CASE fb_state_entry.i16_step OF
(*=======================================================*)
	0:	(* *)
		st_ecd_cmd.enu_cmd := NO_COMMAND;
		st_ecd_cmd.b_job_fehler := FALSE;
		mc_gearindyn_axis.Enable := FALSE;
		mc_gearout_axis.Execute := FALSE;
		mc_camin_axis.Execute := FALSE;
		mc_camout_axis.Execute := FALSE;
		mc_cam_scaleing.Execute := FALSE;
		mc_read_motion_function_point.Execute := FALSE;
		mc_write_motion_function_point.Execute := FALSE;
		mc_read_camtable_slave_dynamics.Execute := FALSE;
		mc_read_camtable_characteristics.Execute := FALSE;
		st_ecd_cmd.meldungen.sm_gear_in_slave := FALSE;
		st_ecd_cmd.meldungen.sm_gear_out_slave := FALSE;
		st_ecd_cmd.meldungen.sm_cam_in_slave := FALSE;
		st_ecd_cmd.meldungen.sm_cam_out_slave := FALSE;
		st_ecd_cmd.meldungen.sm_cam_scaleing_slave := FALSE;
		st_ecd_cmd.meldungen.sm_write_motion_funktion_point := FALSE;
		st_ecd_cmd.meldungen.sm_read_motion_funktion_point := FALSE;
		st_ecd_cmd.meldungen.sm_read_camtable_slave_dynamics := FALSE;
		st_ecd_cmd.meldungen.sm_read_camtable_charakteristik := FALSE;
		st_ecd_cmd.meldungen.sm_camgear_command_timeout := FALSE;

		fb_ton_cmd_timeout.IN := FALSE;
		fb_state_entry.i16_next_step := 10;

(*=======================================================*)
	10:	(* Warte auf Kommando *)
		IF fb_state_entry.E THEN
			st_ecd_cmd.b_job_fehler := FALSE;
			st_ecd_cmd.enu_cmd := NO_COMMAND;
		END_IF

		IF st_ecd_cmd.enu_cmd > NO_COMMAND THEN
			(* Diese Kommandos werden mit Direktsprung ausgeführt, um Zykluszeit zu sparen *)
			IF st_ecd_cmd.enu_cmd = GEAR_IN_SLAVE THEN
				fb_state_entry.i16_next_step := 20;
			ELSIF st_ecd_cmd.enu_cmd = GEAR_OUT_SLAVE THEN
				fb_state_entry.i16_next_step := 30;
			ELSIF st_ecd_cmd.enu_cmd = CAM_IN_SLAVE THEN
				fb_state_entry.i16_next_step := 40;
			ELSIF st_ecd_cmd.enu_cmd = CAM_OUT_SLAVE THEN
				fb_state_entry.i16_next_step := 50;
			ELSIF st_ecd_cmd.enu_cmd = CAM_SCALEING_SLAVE THEN
				fb_state_entry.i16_next_step := 60;
			ELSIF st_ecd_cmd.enu_cmd = READ_MOTION_POINT THEN
				fb_state_entry.i16_next_step := 70;
			ELSIF st_ecd_cmd.enu_cmd = WRITE_MOTION_POINT THEN
				fb_state_entry.i16_next_step := 80;
			ELSIF st_ecd_cmd.enu_cmd = READ_SLAVE_DYNAMICS THEN
				fb_state_entry.i16_next_step := 90;
			ELSIF st_ecd_cmd.enu_cmd = READ_CAMTABLE_CHAR THEN
				fb_state_entry.i16_next_step := 100;
			ELSIF st_ecd_cmd.enu_cmd = RESET THEN
				fb_state_entry.i16_next_step := 999;
			ELSE
				fb_state_entry.i16_next_step := 1000;
			END_IF
		END_IF

(*=======================================================*)
	20:	(* Gear in *)
		fb_ton_cmd_timeout.IN := TRUE;
		mc_gearindyn_axis.Enable := TRUE;
		IF mc_gearindyn_axis.Busy THEN
			fb_state_entry.i16_next_step := 22;
		END_IF

	22:
		IF mc_gearindyn_axis.InGear THEN
			mc_gearindyn_axis.Enable := FALSE;
			fb_state_entry.i16_next_step := 999;
		ELSIF mc_gearindyn_axis.Error THEN
			st_ecd_cmd.meldungen.sm_gear_in_slave := TRUE;
			err_id := mc_gearindyn_axis.ErrorID;
			fb_state_entry.i16_next_step := 1000;
		END_IF

		IF st_ecd_cmd.enu_cmd = GEAR_OUT_SLAVE THEN
			mc_gearindyn_axis.Enable := FALSE;
			fb_ton_cmd_timeout.IN := FALSE;
			fb_ton_vz.IN := FALSE;
			fb_state_entry.i16_next_step := 50;
		END_IF

(*=======================================================*)
	30:	(* Gear out *)
		fb_ton_cmd_timeout.IN := TRUE;
		mc_gearout_axis.Execute := TRUE;
		IF mc_gearout_axis.Busy THEN
			fb_state_entry.i16_next_step := 32;
		END_IF
	32:
		IF NOT mc_gearout_axis.Busy THEN
			mc_gearout_axis.Execute := FALSE;
			IF mc_gearout_axis.Done THEN
				fb_state_entry.i16_next_step := 999;
			ELSIF mc_gearout_axis.Error THEN
				st_ecd_cmd.meldungen.sm_gear_out_slave := TRUE;
				err_id := mc_gearout_axis.ErrorID;
				fb_state_entry.i16_next_step := 1000;
			END_IF
		END_IF

(*=======================================================*)
	40:	(* Cam in *)
		fb_ton_cmd_timeout.IN := NOT st_slaveachse.Status.CamTableQueued;
		mc_camin_axis.Execute := TRUE;
		IF mc_camin_axis.Busy THEN
			fb_state_entry.i16_next_step := 42;
		END_IF
		IF st_ecd_cmd.enu_cmd = CAM_OUT_SLAVE THEN
			mc_camin_axis.Execute := FALSE;
			fb_state_entry.i16_next_step := 50;
		END_IF
	42:
		fb_ton_cmd_timeout.IN := NOT st_slaveachse.Status.CamTableQueued;
		IF NOT mc_camin_axis.Busy THEN
			mc_camin_axis.Execute := FALSE;
			IF mc_camin_axis.InSync THEN
				fb_state_entry.i16_next_step := 999;
			ELSIF mc_camin_axis.Error THEN
				err_id := mc_camin_axis.ErrorID;
				mc_camin_axis.Execute := FALSE;
				st_ecd_cmd.meldungen.sm_cam_in_slave := TRUE;
				fb_state_entry.i16_next_step := 1000;
			END_IF
		END_IF

		IF st_ecd_cmd.enu_cmd = CAM_OUT_SLAVE THEN
			mc_camin_axis.Execute := FALSE;
			fb_ton_cmd_timeout.IN := FALSE;
			fb_ton_vz.IN := FALSE;
			fb_state_entry.i16_next_step := 50;
		END_IF

(*=======================================================*)
	50:	(* Cam out *)
		fb_ton_cmd_timeout.IN := TRUE;
		mc_camout_axis.Execute := TRUE;
		IF mc_camout_axis.Busy THEN
			fb_state_entry.i16_next_step := 52;
		END_IF
	52:
		IF NOT mc_camout_axis.Busy THEN
			mc_camout_axis.Execute := FALSE;
			IF mc_camout_axis.Done THEN
				fb_state_entry.i16_next_step := 999;
			ELSIF mc_camout_axis.Error THEN
				st_ecd_cmd.meldungen.sm_cam_out_slave := TRUE;
				err_id := mc_camout_axis.ErrorID;
				fb_state_entry.i16_next_step := 1000;
			END_IF
		END_IF

(*=======================================================*)
	60:	(* Cam scaleing *)
		fb_ton_cmd_timeout.IN := NOT st_slaveachse.Status.CamScalingPending;
		mc_cam_scaleing.Execute := TRUE;
		IF mc_cam_scaleing.Busy THEN
			fb_state_entry.i16_next_step := 62;
		END_IF
	62:
		fb_ton_cmd_timeout.IN := NOT st_slaveachse.Status.CamScalingPending;
		IF NOT mc_cam_scaleing.Busy THEN
			mc_cam_scaleing.Execute := FALSE;
			IF mc_cam_scaleing.Done THEN
				fb_state_entry.i16_next_step := 999;
			ELSIF mc_cam_scaleing.Error THEN
				st_ecd_cmd.meldungen.sm_cam_scaleing_slave := TRUE;
				err_id := mc_cam_scaleing.ErrorID;
				fb_state_entry.i16_next_step := 1000;
			END_IF
		END_IF

		IF st_ecd_cmd.enu_cmd = CAM_OUT_SLAVE THEN
			mc_cam_scaleing.Execute := FALSE;
			fb_ton_cmd_timeout.IN := FALSE;
			fb_ton_vz.IN := FALSE;
			fb_state_entry.i16_next_step := 50;
		END_IF

(*=======================================================*)
	70:	(* Lesen Motion Funktion Point *)
		fb_ton_cmd_timeout.IN := TRUE;
		mc_read_motion_function_point.Execute := TRUE;
		IF mc_read_motion_function_point.Busy THEN
			fb_state_entry.i16_next_step := 72;
		END_IF
	72:
		IF NOT mc_read_motion_function_point.Busy THEN
			mc_read_motion_function_point.Execute := FALSE;
			IF mc_read_motion_function_point.Done THEN
				fb_state_entry.i16_next_step := 999;
			ELSIF mc_read_motion_function_point.Error THEN
				st_ecd_cmd.meldungen.sm_read_motion_funktion_point := TRUE;
				err_id := mc_read_motion_function_point.ErrorID;
				fb_state_entry.i16_next_step := 1000;
			END_IF
		END_IF

(*=======================================================*)
	80:	(* Schreiben Motion Funktion Point *)
		fb_ton_cmd_timeout.IN := TRUE;
		mc_write_motion_function_point.Execute := TRUE;
		IF mc_write_motion_function_point.Busy THEN
			fb_state_entry.i16_next_step := 82;
		END_IF
	82:
		IF NOT mc_write_motion_function_point.Busy THEN
			mc_write_motion_function_point.Execute := FALSE;
			IF mc_write_motion_function_point.Done THEN
				fb_state_entry.i16_next_step := 999;
			ELSIF mc_write_motion_function_point.Error THEN
				st_ecd_cmd.meldungen.sm_write_motion_funktion_point := TRUE;
				err_id := mc_write_motion_function_point.ErrorID;
				fb_state_entry.i16_next_step := 1000;
			END_IF
		END_IF

(*=======================================================*)
	90:	(* Lesen der Slaveposition in einer Kurvenscheibe *)
		fb_ton_cmd_timeout.IN := TRUE;
		mc_read_camtable_slave_dynamics.Execute := TRUE;
		IF mc_read_camtable_slave_dynamics.Busy THEN
			fb_state_entry.i16_next_step := 92;
		END_IF
	92:
		IF NOT mc_read_camtable_slave_dynamics.Busy THEN
			mc_read_camtable_slave_dynamics.Execute := FALSE;
			IF mc_read_camtable_slave_dynamics.Done THEN
				fb_state_entry.i16_next_step := 999;
			ELSIF mc_read_camtable_slave_dynamics.Error THEN
				st_ecd_cmd.meldungen.sm_write_motion_funktion_point := TRUE;
				err_id := mc_read_camtable_slave_dynamics.ErrorID;
				fb_state_entry.i16_next_step := 1000;
			END_IF
		END_IF

(*=======================================================*)
	100:	(* Lesen der charakteristischen Werte einer Kurvenscheibe *)
		fb_ton_cmd_timeout.IN := TRUE;
		mc_read_camtable_characteristics.Execute := TRUE;
		IF mc_read_camtable_characteristics.Busy THEN
			fb_state_entry.i16_next_step := 102;
		END_IF
	102:
		IF NOT mc_read_camtable_characteristics.Busy THEN
			mc_read_camtable_characteristics.Execute := FALSE;
			IF mc_read_camtable_characteristics.Done THEN
				fb_state_entry.i16_next_step := 999;
			ELSIF mc_read_camtable_characteristics.Error THEN
				st_ecd_cmd.meldungen.sm_read_camtable_charakteristik := TRUE;
				err_id := mc_read_camtable_slave_dynamics.ErrorID;
				fb_state_entry.i16_next_step := 1000;
			END_IF
		END_IF

(*=======================================================*)
	999:	(* Ende - Befehl wurde korrekt abgearbeitet *)
		fb_ton_cmd_timeout.IN := FALSE;
		fb_ton_vz.IN := FALSE;

		mc_gearindyn_axis.Enable := FALSE;
		mc_gearout_axis.Execute := FALSE;
		mc_camin_axis.Execute := FALSE;
		mc_camout_axis.Execute := FALSE;
		mc_cam_scaleing.Execute := FALSE;
		mc_read_motion_function_point.Execute := FALSE;
		mc_write_motion_function_point.Execute := FALSE;
		mc_read_camtable_slave_dynamics.Execute := FALSE;
		mc_read_camtable_characteristics.Execute := FALSE;

		st_ecd_cmd.meldungen.sm_gear_in_slave := FALSE;
		st_ecd_cmd.meldungen.sm_gear_out_slave := FALSE;
		st_ecd_cmd.meldungen.sm_cam_in_slave := FALSE;
		st_ecd_cmd.meldungen.sm_cam_out_slave := FALSE;
		st_ecd_cmd.meldungen.sm_cam_scaleing_slave := FALSE;
		st_ecd_cmd.meldungen.sm_write_motion_funktion_point := FALSE;
		st_ecd_cmd.meldungen.sm_read_motion_funktion_point := FALSE;
		st_ecd_cmd.meldungen.sm_read_camtable_slave_dynamics := FALSE;
		st_ecd_cmd.meldungen.sm_read_camtable_charakteristik := FALSE;
		st_ecd_cmd.meldungen.sm_camgear_command_timeout := FALSE;

		fb_state_entry.i16_next_step := 10;

(*=======================================================*)
	1000: (* Fehler *)
		IF fb_state_entry.E THEN
			st_ecd_cmd.enu_cmd := NO_COMMAND;
			st_ecd_cmd.b_job_fehler := TRUE;
			fb_ton_cmd_timeout.IN := FALSE;
			fb_ton_vz.IN := FALSE;

			mc_gearindyn_axis.Enable := FALSE;
			mc_gearout_axis.Execute := FALSE;
			mc_camin_axis.Execute := FALSE;
			mc_camout_axis.Execute := FALSE;
			mc_cam_scaleing.Execute := FALSE;
			mc_read_motion_function_point.Execute := FALSE;
			mc_write_motion_function_point.Execute := FALSE;
			mc_read_camtable_slave_dynamics.Execute := FALSE;
			mc_read_camtable_characteristics.Execute := FALSE;
		END_IF

		(* Fehler reseten *)
		IF st_ecd_cmd.enu_cmd > ABORT THEN
			st_ecd_cmd.b_job_fehler := FALSE;

			st_ecd_cmd.meldungen.sm_gear_in_slave := FALSE;
			st_ecd_cmd.meldungen.sm_gear_out_slave := FALSE;
			st_ecd_cmd.meldungen.sm_cam_in_slave := FALSE;
			st_ecd_cmd.meldungen.sm_cam_out_slave := FALSE;
			st_ecd_cmd.meldungen.sm_cam_scaleing_slave := FALSE;
			st_ecd_cmd.meldungen.sm_write_motion_funktion_point := FALSE;
			st_ecd_cmd.meldungen.sm_read_motion_funktion_point := FALSE;
			st_ecd_cmd.meldungen.sm_read_camtable_slave_dynamics := FALSE;
			st_ecd_cmd.meldungen.sm_read_camtable_charakteristik := FALSE;
			st_ecd_cmd.meldungen.sm_camgear_command_timeout := FALSE;

			fb_state_entry.i16_next_step := 10;
			err_id :=0;
		END_IF
END_CASE

(* Timeout-Fehler aller Drivekommandos *)
IF fb_ton_cmd_timeout.Q THEN
	fb_ton_cmd_timeout.IN := FALSE;
	st_ecd_cmd.meldungen.sm_camgear_command_timeout := TRUE;
	fb_state_entry.i16_next_step := 1000;
END_IF

(* Statehistory *)
fb_state_entry(
	i16_next_step:= , 
	i16_pos:= 2,
	s_debugtext:= ,
	E=> ,
	X=> , 
	i16_step=> ,
	i16_last_step=> );

fb_cmd_history(i16_current_cmd:= st_ecd_cmd.enu_cmd, last_cmd=> );

(*=============================================================================================*)
(* Ab hier werden alle Cam und Gear Aufträge für eine Achse abgewickelt *)

(* Getriebegleichlauf an der Slaveachse einschalten *)
(* Alternativ kann der Getriebefaktor im Zähler als Fließkommawert angegeben werden, wenn der Nenner 1 ist. *)
mc_gearindyn_axis(
	Enable:= , 
	GearRatio:= r_getriebefaktor,
	Acceleration:= , 
	Deceleration:= , 
	Jerk:= , 
	BufferMode:= mc_buffermode_axis,
	Options:= , 
	Master:= st_masterachse,
	Slave:= st_slaveachse,
	InGear=> , 
	Busy=> , 
	Active=> , 
	CommandAborted=> , 
	Error=> , 
	ErrorID=> );

(*=============================================================================================*)
(* Getriebegleichlauf ausschalten *)
mc_gearout_axis(
	Execute:= ,
	Options:= ,
	Slave:= st_slaveachse,
	Done=> ,
	Busy=> ,
	Error=> ,
	ErrorID=> );

(*=============================================================================================*)
(* Kurvenscheibe am Slave aktivieren *)
mc_camin_axis(
	Execute:= , 
	ActivationMode:= mc_activation_mode_camin,
	ActivationPosition:= lr_activation_position_camin,
	CamTableID:= mc_cam_table_id,
	Scaling:= st_camscaling_data,
	Options:= st_camin_options,
	Master:= st_masterachse,
	Slave:= st_slaveachse,
	InSync=> , 
	Busy=> , 
	Active=> , 
	CommandAborted=> , 
	Error=> ,
	ErrorID=> );

(*=============================================================================================*)
(* Kurvenscheibe ausschalten *)
mc_camout_axis(
	Execute:= ,
	Slave:= st_slaveachse,
	Options:= ,
	Done=> ,
	Busy=> ,
	Error=> ,
	ErrorID=> );

(*=============================================================================================*)
(* Scalierung einer Kurvenscheibe *)
mc_cam_scaleing(
	Execute:= , 
	ActivationMode:= mc_activation_mode_scaleing,
	ActivationPosition:= lr_activation_position_scaleing,
	CamTableID:= mc_cam_table_id,
	Scaling:= st_camscaling_data,
	Options:= ,
	Slave:= st_slaveachse,
	Done=> , 
	Busy=> ,
	Active=> , 
	CommandAborted=> ,
	Error=> , 
	ErrorID=> );

(*=============================================================================================*)
(* Lesen eines Punktes in der Kurvenscheibe *)
mc_read_motion_function_point(
	Execute:= ,
	CamTableID:= mc_cam_table_id,
	PointID:= mc_cam_point_id,
	Point:= mc_motion_function_point,
	Done=> , 
	Busy=> , 
	Error=> , 
	ErrorID=> );

(*=============================================================================================*)
(* Verändern von einem Punkt in der Kurvenscheibe *)
mc_write_motion_function_point(
	Execute:= , 
	CamTableID:= mc_cam_table_id,
	PointID:= mc_cam_point_id,
	Point:= mc_motion_function_point,
	Done=> , 
	Busy=> , 
	Error=> ,
	ErrorID=> );

(*=============================================================================================*)
(* Lesen einer Slaveposition in der Kurvenscheibe *)
mc_read_camtable_slave_dynamics(
	Execute:= ,
	CamTableID:= mc_cam_table_id,
	MasterPosition:= r_master_position,
	Done=> , 
	Busy=> ,
	Error=> , 
	ErrorID=> ,
	SlavePosition=> , 
	SlaveVelocity=> , 
	SlaveAcceleration=> );

(*=============================================================================================*)
(* Lesen der charakteristischen Werte einer Kurvenscheibe *)
mc_read_camtable_characteristics(
	Execute:= , 
	CamTableID:= mc_cam_table_id,
	CamTableCharac:= st_cam_table_characteristics,
	Done=> , 
	Busy=> , 
	Error=> , 
	ErrorID=> );
END_FUNCTION_BLOCK

(* POU EPT Lib/Funktionsbausteine/ST_BerechnungOverride, ST *)
FUNCTION_BLOCK ST_BerechnungOverride
VAR_INPUT
	i16_betriebsart				: enum_betriebsarten;
	lr_skalierung_slave_achse1		: LREAL;
	lr_skalierung_slave_achse2		: LREAL;
	lr_override_vorgabe			: LREAL;
	lr_faktor						: LREAL;

	lr_FaktorHub				: LREAL;
	lr_HubAuto					: LREAL;
END_VAR
VAR_OUTPUT
	lr_override					: LREAL := 0.0;
END_VAR
VAR
	lr_offset						: LREAL := 100.0;
	tmp_lr_override_slave1		: LREAL := 0.0;
	tmp_lr_override_slave2		: LREAL := 0.0;

	lr_ProzentDerRichtdrehzahl	: LREAL;
	lr_Reduzierung				: LREAL;
END_VAR
(* Funktion zur Berechnung des Override der  Masterachse: y = - faktor * x^2 + offset *)
(* Die Funktion besteht aus einer auf dem Kopf stehenden Parabel, welche um den faktor nach oben verschoben ist *)
(* Aufpassen bei den Nullstellen der Funktion, wenn faktor und offset verändert werden *)

(* Die Anpassung der maximalen Mastergeschwindigkeit an die Verfahrlänge des Slaves wird hier einfach über eine empirisch ermittelte Funktion realisiert *)
(* Eine verbesserte Anpassung stellt die Berechnung der maximalen Mastergeschwindigkeit (ST_MFMaxMasterVelo) im CamEditor dar. *)

tmp_lr_override_slave1 := - lr_faktor * (lr_skalierung_slave_achse1 * lr_skalierung_slave_achse1)  + lr_offset;
tmp_lr_override_slave2 := - lr_faktor * (lr_skalierung_slave_achse2 * lr_skalierung_slave_achse2)  + lr_offset;

IF tmp_lr_override_slave1 < 0.0 THEN
	 tmp_lr_override_slave1 := 0.0;
ELSIF tmp_lr_override_slave1 >= 100.0 THEN
	 tmp_lr_override_slave1 := 100.0;
END_IF
IF tmp_lr_override_slave2 < 0.0 THEN
	 tmp_lr_override_slave2 := 0.0;
ELSIF tmp_lr_override_slave2 >= 100.0 THEN
	 tmp_lr_override_slave2 := 100.0;
END_IF

IF i16_betriebsart = AUTO THEN
	(* Nur wenn der mit der Funktion berechnete Override kleiner ist, als die Vorgabe, dann wird der Funktionswert übernommen *)
	IF 	tmp_lr_override_slave1 < lr_override_vorgabe OR
		tmp_lr_override_slave2 < lr_override_vorgabe THEN

		IF tmp_lr_override_slave1 <= tmp_lr_override_slave2 THEN
			lr_override := tmp_lr_override_slave1;
		ELSIF tmp_lr_override_slave2 < tmp_lr_override_slave1 THEN
			lr_override := tmp_lr_override_slave2;
		ELSE
			lr_override := lr_override_vorgabe;
		END_IF

	ELSE
		lr_override := lr_override_vorgabe;
	END_IF
ELSE
	lr_override := lr_override_vorgabe;
END_IF


(*neue Berechnung==========================================================================*)
(*Reduzierung abhängig von der Nenndrehzahl*)
lr_ProzentDerRichtdrehzahl:=(lr_HubAuto *100)/250;
IF	lr_HubAuto >250 AND
	lr_override_vorgabe > lr_override THEN
	lr_override := 100-((lr_override_vorgabe - lr_override) * (lr_ProzentDerRichtdrehzahl /100)) ;
END_IF

(*nur Reduzieren wenn das Ergebniss kleiner ist als bei der Reduzierung durch die Pin Anzahl*)
lr_Reduzierung:= (lr_override_vorgabe - lr_override)/100;
IF	(1 - lr_Reduzierung) < lr_FaktorHub THEN
	lr_override := lr_override;
ELSE
	lr_override:= 100 * lr_FaktorHub;
END_IF

IF	lr_override > lr_override_vorgabe OR
	lr_override < 0 THEN
	lr_override:= lr_override_vorgabe;
END_IF

(*Beim Einfädeln wird der Override vom Bausstein ST_TippTasten einfach durchgeschleust*)
IF	ST_TippTasten.b_einfaedeln_aktiv OR
	ST_TippTasten.b_initialisierungsphase THEN
	lr_override := lr_override_vorgabe;
END_IF

(*bei Prüfteilen Override fest auf 30% *)
IF	lr_override_vorgabe > 30 AND
	(FIND( gst_datensatz.st_md.s_aktuelle_artikelnummer,'ruef') <> 0 OR FIND( gst_datensatz.st_md.s_aktuelle_artikelnummer,'erth') <> 0)THEN
	lr_override := 30;
END_IF
END_FUNCTION_BLOCK

(* POU Gemeinsamkeiten17xx/Bedienen/ST_TippTasten, ST *)
PROGRAM ST_TippTasten
VAR_INPUT
	(* Geschwindigkeit / Stufe *)
	i16_akt_stufe						: INT := 0;	(* 0-9 *)
	b_initialisierungsphase				: BOOL := FALSE;
	b_einfaedeln_aktiv				: BOOL := FALSE;
END_VAR
VAR_IN_OUT
	st_visu							: struct_visu;
	st_visu_hinten						: struct_visu_hinten;
END_VAR
VAR
	lr_override						: LREAL := 25;
	lr_override_gestuft					: LREAL := 10;
	r_trig_tippen						: R_TRIG;
	r_trig_tippen_einfaedeln			: R_TRIG;
	r_trig_vorgabe					: R_TRIG;
	b_freigabe_override_auto			: BOOL := FALSE;
	fb_r_trig_quittieren					: R_TRIG;
END_VAR

VAR CONSTANT
	lr_override_init_einfaedel			: LREAL := 25;
END_VAR
(* Mit den zeitlichen Impulsen vom Handrad lässt sich der Override aller Achsen verändern. Die Geschwindigkeit wird im "ST_AxisJobCtrl_Motion" limitiert. *)
(* Tipp-Taste *)

r_trig_tippen(
		CLK:=NOT b_einfaedeln_aktiv AND (st_visu.b_tippen_start OR visu_hinten.out.b_start OR ST_Euchner_Handbedienpult.b_Taste_Power),
		Q=> );
r_trig_tippen_einfaedeln(
		CLK:= b_einfaedeln_aktiv AND (st_visu_hinten.out.b_tippen OR ST_Euchner_Handbedienpult.b_Taste_Power),
		Q=> );
r_trig_vorgabe(
		CLK:= st_visu.b_geschwindigkeit_vorgabe, Q=> );

(* Flanken *)
fb_r_trig_quittieren(CLK:= st_visu.b_quittieren OR st_visu_hinten.out.b_quittieren, Q=> );

CASE gi16_betriebsart OF
	AUTO:
		gb_ba_auto_kontroller := TRUE;

		IF r_trig_tippen.Q OR fb_r_trig_quittieren.Q THEN
			b_freigabe_override_auto := TRUE;
		END_IF

		IF b_einfaedeln_aktiv OR b_initialisierungsphase THEN
			lr_override := lr_override_gestuft := lr_override_init_einfaedel;
		ELSE

			IF r_trig_vorgabe.Q THEN
				i16_akt_stufe := 9;
			END_IF
			IF b_freigabe_override_auto THEN
				(* Override für Achsen mit "Vollgas" im Automatikbetrieb *)
				lr_override := 100;
				(* Override für Achsen, welche in Abstufung gefahren werden *)
				IF  i16_akt_stufe>= 0 AND i16_akt_stufe<= 9 THEN
					(* Overridevorgabe im Automatikbetrieb *)
					lr_override_gestuft := (i16_akt_stufe +1) * 10;
				ELSE
					(* Falls Geschwindigkeitsstufe was anderes als 0-9 enthält: Override auf 0: Keine Achse fährt *)
					lr_override_gestuft := 0;
				END_IF
			ELSE
				lr_override := lr_override_gestuft := 0;
			END_IF
		END_IF

	TIPPEN:
		b_freigabe_override_auto := FALSE;

		IF r_trig_tippen.Q OR lr_override > 0 OR  lr_override_gestuft > 0 THEN
			gb_ba_auto_kontroller := TRUE;
		ELSE
			gb_ba_auto_kontroller := FALSE;
		END_IF

		IF ST_Euchner_Handbedienpult.i16_Handrad_delta > 0 THEN
			lr_override := lr_override_gestuft := ABS(ST_Euchner_Handbedienpult.i16_Handrad_delta) * 0.1;
		ELSE
			lr_override := lr_override_gestuft := 0;
		END_IF

	HAND:
		gb_ba_auto_kontroller := FALSE;
		b_freigabe_override_auto := FALSE;
		lr_override := lr_override_gestuft := ABS(ST_Euchner_Handbedienpult.i16_Handrad_delta)* 0.1;
END_CASE

(* Abfrage maximaler Override grösser 100% *)
IF lr_override > 100 THEN
	lr_override := 100;
END_IF
IF lr_override_gestuft > 100 THEN
	lr_override_gestuft := 100;
END_IF
END_PROGRAM

(* POU Gemeinsamkeiten17xx/Bedienen/ST_Euchner_Handbedienpult, ST *)
PROGRAM ST_Euchner_Handbedienpult
VAR
	(* Eingänge von der Hardware *)
	e_Taste_Zustimm			AT %I* : BOOL;
	e_Taste_Plus				AT %I* : BOOL;
	e_Taste_Power			AT %I* : BOOL;
	e_Taste_Minus			AT %I* : BOOL;

	e_i16_Zaehler			AT %I* : INT;

	(* Instanzen *)
	fb_ton					: TON;

	(* Merker *)
	i16_merkpos				: INT := 0;
END_VAR
VAR_OUTPUT
	b_Taste_Zustimm			: BOOL := FALSE;
	b_Taste_Plus				: BOOL := FALSE;
	b_Taste_Power			: BOOL := FALSE;
	b_Taste_Minus			: BOOL := FALSE;

	i16_Handrad_delta		: INT := 0;
END_VAR
(* Tasten *)
b_Taste_Zustimm	:= e_Taste_Zustimm;
b_Taste_Plus	:= e_Taste_Plus;
b_Taste_Power := e_Taste_Power;
b_Taste_Minus := e_Taste_Minus;

(* Generiere Impuls für Delta Zähler *)
fb_ton(IN:= NOT fb_ton.Q , PT:= t#100ms, Q=> , ET=> );

IF fb_ton.Q THEN
	i16_Handrad_delta := e_i16_Zaehler - i16_merkpos;
	i16_merkpos := e_i16_Zaehler;
END_IF
END_PROGRAM

(* POU Rasterfolie/ST_Rasterfolieneinzug, ST *)
PROGRAM ST_Rasterfolieneinzug
VAR_INPUT
	st_config							: struct_config;
	st_ctrl_in							: struct_ctrl_in;
END_VAR
VAR_IN_OUT
	st_visu							: struct_visu;
END_VAR
VAR_OUTPUT
	st_ctrl_out						: struct_ctrl_out;
END_VAR
VAR
	fb_ton_wz						: TON;
	fb_ton_uez						: TON;
	fb_ton_quitt						: TON;
	fb_ton_gls_rafo_vorhanden		: TON;
	fb_tof_gls_rafo_ende			: TOF;
	fb_tof_AbschaltungIonisierung		: TOF;
	fb_r_trig_start						: R_TRIG;
	fb_r_trig_vorschubkontrolle			: R_TRIG;
	fb_f_trig_vorschubkontrolle			: F_TRIG;
	fb_state_entry						: ST_StateEntry;
	i								: INT := 0;
	sm_fehler_rafo_vorschub			: BOOL := FALSE;
	sm_keine_rafo_im_einzug		: BOOL := FALSE;

	e_rasfo_ende						AT %I* : BOOL;
	e_rasfo_vorschubkontrolle			AT %I* : BOOL;
	e_rasfo_rueckzugueberwachung		AT %I* : BOOL;

	(* Ausgang Ionisierung Rasterfolie einschalten *)
	aIonisierungEin				AT %Q* : BOOL;

END_VAR
(* Zeiten *)
fb_ton_wz(IN:= , PT:= , Q=>  , ET=> );
fb_ton_uez(IN:= , PT:= t#1000ms, Q=>  , ET=> );
fb_ton_quitt(IN:= , PT:= t#100ms, Q=> , ET=> );
fb_ton_gls_rafo_vorhanden(IN:= e_rasfo_ende, PT:= T#300ms, Q=> , ET=> );
fb_tof_gls_rafo_ende(IN:= fb_ton_gls_rafo_vorhanden.Q, PT:= T#300ms, Q=> , ET=> );
fb_tof_AbschaltungIonisierung(IN:= fb_state_entry.i16_step = 200, PT:= T#2m, Q=> , ET=> );

(* Flanken *)
fb_r_trig_start(CLK:= st_ctrl_in.b_start, Q=> );
fb_r_trig_vorschubkontrolle(CLK:= e_rasfo_vorschubkontrolle, Q=> );
fb_f_trig_vorschubkontrolle(CLK:= e_rasfo_vorschubkontrolle, Q=> );


(* Steuerung Ionisierung *)
IF gi16_maschinenstatusinfo = STATUS_MASCHINE_ARBEITET THEN
	aIonisierungEin := fb_tof_AbschaltungIonisierung.Q;
ELSE
	aIonisierungEin := FALSE;
END_IF


(* Toplevel *)
IF fb_state_entry.i16_next_step > INIT AND fb_state_entry.i16_next_step < FEHLER THEN
	IF fb_state_entry.i16_next_step < STOP THEN
		IF st_ctrl_in.b_stop THEN
			fb_state_entry.i16_next_step := STOP;
		END_IF
	END_IF
	(* Allgemeine Fehler *)
	IF	zyl_rafo_faenger.st_ctrl.out.b_fehler OR
		zyl_rafo_klemmen.st_ctrl.out.b_fehler OR
		zyl_rafo_vorschub.st_ctrl.out.b_fehler
		THEN
			fb_state_entry.i16_next_step := FEHLER;

	(* Zylinder im Handbetrieb *)
	ELSIF	gi16_betriebsart = HAND AND (
			(st_visu.st_zyl.i16_nr_zyl_im_handbetrieb = zyl_rafo_faenger.fb.st_config.i16_identnummer) OR
			(st_visu.st_zyl.i16_nr_zyl_im_handbetrieb = zyl_rafo_klemmen.fb.st_config.i16_identnummer) OR
			(st_visu.st_zyl.i16_nr_zyl_im_handbetrieb = zyl_rafo_vorschub.fb.st_config.i16_identnummer) )
			THEN
				fb_state_entry.i16_next_step := FEHLER;
	END_IF
END_IF

sm_keine_rafo_im_einzug:=ST_Z_Achse.sm_keine_rafo_im_einzug;

(* ======================================Schrittkette======================================== *)
fb_state_entry(
	i16_next_step:= ,
	i16_pos:= 1,
	s_debugtext:= ,
	E=> ,
	X=> , 
	i16_step=> ,
	i16_last_step=> );

CASE fb_state_entry.i16_step OF
(*=======================================================*)
	INIT_OBJ:
		IF st_config.b_config_fertig THEN
			fb_state_entry.i16_next_step := INIT;
		END_IF

(*=======================================================*)
	INIT:
		IF fb_state_entry.E THEN
			fb_ton_wz.IN := FALSE;
			fb_ton_uez.IN := FALSE;
			fb_ton_quitt.IN := FALSE;
			st_ctrl_out.b_fehler := FALSE;
			st_ctrl_out.b_bereit := FALSE;
			st_ctrl_out.b_fertig := FALSE;
			zyl_rafo_faenger.st_ctrl.in.b_ausfahren := FALSE;
			zyl_rafo_faenger.st_ctrl.in.b_einfahren := FALSE;
			zyl_rafo_klemmen.st_ctrl.in.b_ausfahren := FALSE;
			zyl_rafo_klemmen.st_ctrl.in.b_einfahren := FALSE;
			zyl_rafo_vorschub.st_ctrl.in.b_ausfahren := FALSE;
			zyl_rafo_vorschub.st_ctrl.in.b_einfahren := FALSE;
			sm_fehler_rafo_vorschub := FALSE;
			sm_keine_rafo_im_einzug := FALSE;
		END_IF

		(*-----------------------Weiterschaltbedingungen----------------------------*)
		IF st_ctrl_in.b_init THEN
			zyl_rafo_faenger.st_ctrl.in.b_quittieren := FALSE;
			zyl_rafo_klemmen.st_ctrl.in.b_quittieren := FALSE;
			zyl_rafo_vorschub.st_ctrl.in.b_quittieren := FALSE;
			IF gst_datensatz.st_md.b_wt_transport_simulation THEN
				fb_state_entry.i16_next_step := BEREIT;
			ELSE
				fb_state_entry.i16_next_step := 20;
			END_IF
		END_IF

(*=======================================================*)
	20:	(* Klemmung ausfahren und Folie halten *)
		IF fb_state_entry.E THEN
			zyl_rafo_klemmen.st_ctrl.in.b_ausfahren := TRUE;
		END_IF

		(*-----------------------Weiterschaltbedingungen----------------------------*)
		IF zyl_rafo_klemmen.st_ctrl.out.b_ausgefahren THEN
			zyl_rafo_klemmen.st_ctrl.in.b_ausfahren := FALSE;
			fb_state_entry.i16_next_step := 30;
		END_IF

(*=======================================================*)
	30:	(* Fänger einfahren *)
		IF fb_state_entry.E THEN
			zyl_rafo_faenger.st_ctrl.in.b_einfahren := TRUE;
		END_IF

		(*-----------------------Weiterschaltbedingungen----------------------------*)
		IF zyl_rafo_faenger.st_ctrl.out.b_eingefahren THEN
			zyl_rafo_faenger.st_ctrl.in.b_einfahren := FALSE;
			fb_state_entry.i16_next_step := 40;
		END_IF

(*=======================================================*)
	40:	(* Vorschub zurück fahren *)
		IF fb_state_entry.E THEN
			zyl_rafo_vorschub.st_ctrl.in.b_einfahren := TRUE;
		END_IF

		(*-----------------------Weiterschaltbedingungen----------------------------*)
		IF zyl_rafo_vorschub.st_ctrl.out.b_eingefahren THEN
			zyl_rafo_vorschub.st_ctrl.in.b_einfahren := FALSE;
			fb_state_entry.i16_next_step := 50;
		END_IF

(*=======================================================*)
	50:	(* Fänger ausfahren *)
		IF fb_state_entry.E THEN
			zyl_rafo_faenger.st_ctrl.in.b_ausfahren := TRUE;
		END_IF

		(*-----------------------Weiterschaltbedingungen----------------------------*)
		IF zyl_rafo_faenger.st_ctrl.out.b_ausgefahren THEN
			zyl_rafo_faenger.st_ctrl.in.b_ausfahren := FALSE;
			fb_state_entry.i16_next_step := 60;
		END_IF

(*=======================================================*)
	60:	(* Klemmung einfahren *)
		IF fb_state_entry.E THEN
			zyl_rafo_klemmen.st_ctrl.in.b_einfahren := TRUE;
		END_IF

		(*-----------------------Weiterschaltbedingungen----------------------------*)
		IF zyl_rafo_klemmen.st_ctrl.out.b_eingefahren THEN
			zyl_rafo_klemmen.st_ctrl.in.b_einfahren := FALSE;
			fb_state_entry.i16_next_step := BEREIT;
		END_IF

(*=======================================================*)
	BEREIT:
		IF fb_state_entry.E THEN
			st_ctrl_out.b_bereit := TRUE;
			st_ctrl_out.b_fertig := TRUE;
		END_IF

		(*-----------------------Weiterschaltbedingungen----------------------------*)
		IF st_ctrl_in.b_start THEN
			st_ctrl_out.b_fertig := FALSE;
			fb_state_entry.i16_next_step := 110;
		END_IF

(*=======================================================*)
	110:	(* Prüfe Rasterfolie im Einzug *)		(*wird im BEREIT der Z-Achse geprütf*)

		fb_state_entry.i16_next_step := 200;

(*===========================Vorschub Folie============================*)
	200:	(* Vorschub ausfahren und Vorschub prüfen *)
		IF fb_state_entry.E THEN
			zyl_rafo_vorschub.st_ctrl.in.b_ausfahren := TRUE;
		END_IF

		(*-----------------------Weiterschaltbedingungen----------------------------*)
		(* Vorschubkontrolle durch positive Flanke *)
		IF fb_r_trig_vorschubkontrolle.Q THEN
			fb_state_entry.i16_next_step := 210;
		ELSIF zyl_rafo_vorschub.st_ctrl.out.b_ausgefahren THEN
			sm_fehler_rafo_vorschub := TRUE;
			fb_state_entry.i16_next_step := FEHLER;
		END_IF

(*=======================================================*)
	210:	(* Verhindere Signalüberschneidungen *)
		IF fb_state_entry.E THEN
			fb_ton_wz.PT := t#1000ms;
 			fb_ton_wz.IN := TRUE;
		END_IF

		(*-----------------------Weiterschaltbedingungen----------------------------*)
		(* Vorschubkontrolle durch negative Flanke *)
		IF fb_f_trig_vorschubkontrolle.Q THEN
			fb_ton_wz.IN := FALSE;
			fb_state_entry.i16_next_step := 220;
		ELSIF zyl_rafo_vorschub.st_ctrl.out.b_ausgefahren AND fb_ton_wz.Q THEN
			sm_fehler_rafo_vorschub := TRUE;
			fb_state_entry.i16_next_step := FEHLER;
		END_IF

(*=======================================================*)
	220:	(* Vorschub ist fertig ausgefahren *)

		(*-----------------------Weiterschaltbedingungen----------------------------*)
		IF zyl_rafo_vorschub.st_ctrl.out.b_ausgefahren AND gb_ba_auto_kontroller THEN
			zyl_rafo_vorschub.st_ctrl.in.b_ausfahren := FALSE;
			fb_state_entry.i16_next_step := 230;
		END_IF

(*=======================================================*)
	230:	(* Klemmung ausfahren und Folie halten *)
		IF fb_state_entry.E THEN
			zyl_rafo_klemmen.st_ctrl.in.b_ausfahren := TRUE;
		END_IF

		(*-----------------------Weiterschaltbedingungen----------------------------*)
		IF zyl_rafo_klemmen.st_ctrl.out.b_ausgefahren AND gb_ba_auto_kontroller THEN
			zyl_rafo_klemmen.st_ctrl.in.b_ausfahren := FALSE;
			fb_state_entry.i16_next_step := 240;
		END_IF

(*=======================================================*)
	240:	(* Fänger einfahren *)
		IF fb_state_entry.E THEN
			zyl_rafo_faenger.st_ctrl.in.b_einfahren := TRUE;
		END_IF

		(*-----------------------Weiterschaltbedingungen----------------------------*)
		IF zyl_rafo_faenger.st_ctrl.out.b_eingefahren AND gb_ba_auto_kontroller THEN
			zyl_rafo_faenger.st_ctrl.in.b_einfahren := FALSE;
			fb_state_entry.i16_next_step := 250;
		END_IF

(*=======================================================*)
	250:	(* Vorschub zurück fahren *)
		IF fb_state_entry.E THEN
			zyl_rafo_vorschub.st_ctrl.in.b_einfahren := TRUE;
		END_IF

		(*-----------------------Weiterschaltbedingungen----------------------------*)
		IF zyl_rafo_vorschub.st_ctrl.out.b_eingefahren AND gb_ba_auto_kontroller THEN
			zyl_rafo_vorschub.st_ctrl.in.b_einfahren := FALSE;
			fb_state_entry.i16_next_step := 260;
		END_IF

(*=======================================================*)
	260: (* Warte *)
		IF fb_state_entry.E THEN
			fb_ton_wz.PT := t#300ms;
 			fb_ton_wz.IN := TRUE;
		END_IF

		(*-----------------------Weiterschaltbedingungen----------------------------*)
		IF fb_ton_wz.Q THEN
			fb_ton_wz.IN := FALSE;
			(* Rasterfolieneinzug lüften
			Dies wird nur gemacht, wenn die Nocken ungleich 0 sind und Anfangs- und Endnocke aunterschiedlich sind
			Zwischen den Nocken wird die Rasterfolie vom Werkzeug gehalten *)
			IF gst_datensatz.st_wkz.nockenschaltwerk_bestueckachse.arr_nocken[NO_RASTERFOLIE_LUEFTEN].r_cam_begin <> 0 AND
				gst_datensatz.st_wkz.nockenschaltwerk_bestueckachse.arr_nocken[NO_RASTERFOLIE_LUEFTEN].r_cam_begin <> gst_datensatz.st_wkz.nockenschaltwerk_bestueckachse.arr_nocken[NO_RASTERFOLIE_LUEFTEN].r_cam_end THEN
				fb_state_entry.i16_next_step := 290;(* Ablauf mit Lüften *)
			ELSE
				fb_state_entry.i16_next_step := 270;(* Ablauf ohne Lüften *)
			END_IF
		END_IF

(*=======================================================*)
	270:	(* Fänger ausfahren *)
		IF fb_state_entry.E THEN
			zyl_rafo_faenger.st_ctrl.in.b_ausfahren := TRUE;
		END_IF

		(*-----------------------Weiterschaltbedingungen----------------------------*)
		IF zyl_rafo_faenger.st_ctrl.out.b_ausgefahren AND gb_ba_auto_kontroller THEN
			zyl_rafo_faenger.st_ctrl.in.b_ausfahren := FALSE;
			fb_state_entry.i16_next_step := 280;
		END_IF

(*=======================================================*)
	280:	(* Klemmung einfahren *)
		IF fb_state_entry.E THEN
			zyl_rafo_klemmen.st_ctrl.in.b_einfahren := TRUE;
		END_IF

		(*-----------------------Weiterschaltbedingungen----------------------------*)
		IF zyl_rafo_klemmen.st_ctrl.out.b_eingefahren AND gb_ba_auto_kontroller THEN
			zyl_rafo_klemmen.st_ctrl.in.b_einfahren := FALSE;
			fb_state_entry.i16_next_step := 290;
		END_IF

(*=======================================================*)
	290:	(* Bandüberstand nach WKZ prüfen und eventuell zurückziehen *)

		(*-----------------------Weiterschaltbedingungen----------------------------*)
		IF e_rasfo_rueckzugueberwachung THEN
			fb_state_entry.i16_next_step := 300;
		ELSE
			fb_state_entry.i16_next_step := BEREIT;
		END_IF

(*===========================Rückzug Folie============================*)
	300:	(* Klemmung ausfahren und Folie halten *)
		IF fb_state_entry.E THEN
			zyl_rafo_klemmen.st_ctrl.in.b_ausfahren := TRUE;
		END_IF

		(*-----------------------Weiterschaltbedingungen----------------------------*)
		IF zyl_rafo_klemmen.st_ctrl.out.b_ausgefahren AND gb_ba_auto_kontroller THEN
			zyl_rafo_klemmen.st_ctrl.in.b_ausfahren := FALSE;
			fb_state_entry.i16_next_step := 310;
		END_IF

(*=======================================================*)
	310:	(* Fänger einfahren *)
		IF fb_state_entry.E THEN
			zyl_rafo_faenger.st_ctrl.in.b_einfahren := TRUE;
		END_IF

		(*-----------------------Weiterschaltbedingungen----------------------------*)
		IF zyl_rafo_faenger.st_ctrl.out.b_eingefahren AND gb_ba_auto_kontroller THEN
			zyl_rafo_faenger.st_ctrl.in.b_einfahren := FALSE;
			fb_state_entry.i16_next_step := 320;
		END_IF

(*=======================================================*)
	320:	(* Vorschub ausfahren *)
		IF fb_state_entry.E THEN
			zyl_rafo_vorschub.st_ctrl.in.b_ausfahren := TRUE;
		END_IF

		(*-----------------------Weiterschaltbedingungen----------------------------*)
		IF zyl_rafo_vorschub.st_ctrl.out.b_ausgefahren AND gb_ba_auto_kontroller THEN
			zyl_rafo_vorschub.st_ctrl.in.b_ausfahren := FALSE;
			fb_state_entry.i16_next_step := 330;
		END_IF

(*=======================================================*)
	330:	(* Fänger ausfahren *)
		IF fb_state_entry.E THEN
			zyl_rafo_faenger.st_ctrl.in.b_ausfahren := TRUE;
		END_IF

		(*-----------------------Weiterschaltbedingungen----------------------------*)
		IF zyl_rafo_faenger.st_ctrl.out.b_ausgefahren AND gb_ba_auto_kontroller THEN
			zyl_rafo_faenger.st_ctrl.in.b_ausfahren := FALSE;
			fb_state_entry.i16_next_step := 340;
		END_IF

(*=======================================================*)
	340:	(* Klemmung einfahren *)
		IF fb_state_entry.E THEN
			zyl_rafo_klemmen.st_ctrl.in.b_einfahren := TRUE;
		END_IF

		(*-----------------------Weiterschaltbedingungen----------------------------*)
		IF zyl_rafo_klemmen.st_ctrl.out.b_eingefahren AND gb_ba_auto_kontroller THEN
			zyl_rafo_klemmen.st_ctrl.in.b_einfahren := FALSE;
			fb_state_entry.i16_next_step := 350;
		END_IF

(*=======================================================*)
	350:	(* Vorschub zurück fahren *)
		IF fb_state_entry.E THEN
			zyl_rafo_vorschub.st_ctrl.in.b_einfahren := TRUE;
		END_IF

		(*-----------------------Weiterschaltbedingungen----------------------------*)
		IF zyl_rafo_vorschub.st_ctrl.out.b_eingefahren AND gb_ba_auto_kontroller THEN
			zyl_rafo_vorschub.st_ctrl.in.b_einfahren := FALSE;
			fb_state_entry.i16_next_step := 290;
		END_IF

(*=======================================================*)
	FEHLER:
		IF fb_state_entry.E THEN
			st_ctrl_out.b_fehler := TRUE;
			fb_ton_quitt.IN := FALSE;
			zyl_rafo_faenger.st_ctrl.in.b_quittieren := FALSE;
			zyl_rafo_klemmen.st_ctrl.in.b_quittieren := FALSE;
			zyl_rafo_vorschub.st_ctrl.in.b_quittieren := FALSE;
		END_IF

		(*-----------------------Weiterschaltbedingungen----------------------------*)
		IF st_ctrl_in.b_quitt AND NOT fb_state_entry.E THEN
			st_ctrl_out.b_fehler := FALSE;
			zyl_rafo_faenger.st_ctrl.in.b_quittieren := TRUE;
			zyl_rafo_klemmen.st_ctrl.in.b_quittieren := TRUE;
			zyl_rafo_vorschub.st_ctrl.in.b_quittieren := TRUE;
			fb_ton_quitt.IN := TRUE;
		END_IF

		IF fb_ton_quitt.Q THEN
			fb_ton_quitt.IN := FALSE;
			fb_state_entry.i16_next_step := INIT;
		END_IF

(*=======================================================*)
	STOP:
		IF fb_state_entry.E THEN
			fb_ton_quitt.IN := FALSE;
		END_IF

		(*-----------------------Weiterschaltbedingungen----------------------------*)
		IF st_ctrl_in.b_quitt AND NOT fb_state_entry.E THEN
			fb_ton_quitt.IN := TRUE;
		END_IF

		IF fb_ton_quitt.Q THEN
			fb_ton_quitt.IN := FALSE;
			fb_state_entry.i16_next_step := INIT;
		END_IF
END_CASE

fb_state_entry(
	i16_next_step:= , 
	i16_pos:= 2,
	s_debugtext:= ,
	E=> , 
	X=> , 
	i16_step=> ,
	i16_last_step=> );

IF st_config.b_config_fertig THEN
	(* Fehlermeldungen und Betriebsmeldungen ab dem Startindex in die globalen Meldungsarrays schreiben *)
	garr_stoermeldungen[st_config.i16_meld_startindex + 0] := sm_fehler_rafo_vorschub;
	garr_stoermeldungen[st_config.i16_meld_startindex + 1] := sm_keine_rafo_im_einzug;
	garr_stoermeldungen[st_config.i16_meld_startindex + 2] := FALSE;
	garr_stoermeldungen[st_config.i16_meld_startindex + 3] := FALSE;
	garr_stoermeldungen[st_config.i16_meld_startindex + 4] := FALSE;
	garr_stoermeldungen[st_config.i16_meld_startindex + 5] := FALSE;
	garr_stoermeldungen[st_config.i16_meld_startindex + 6] := FALSE;
	garr_stoermeldungen[st_config.i16_meld_startindex + 7] := FALSE;
	garr_stoermeldungen[st_config.i16_meld_startindex + 8] := FALSE;
	garr_stoermeldungen[st_config.i16_meld_startindex + 9] := FALSE;
	garr_stoermeldungen[st_config.i16_meld_startindex + 10] := FALSE;
	garr_stoermeldungen[st_config.i16_meld_startindex + 11] := FALSE;
	garr_stoermeldungen[st_config.i16_meld_startindex + 12] := FALSE;
	garr_stoermeldungen[st_config.i16_meld_startindex + 13] := FALSE;
	garr_stoermeldungen[st_config.i16_meld_startindex + 14] := FALSE;
	garr_stoermeldungen[st_config.i16_meld_startindex + 15] := FALSE;
	garr_stoermeldungen[st_config.i16_meld_startindex + 16] := FALSE;
	garr_stoermeldungen[st_config.i16_meld_startindex + 17] := FALSE;
	garr_stoermeldungen[st_config.i16_meld_startindex + 18] := FALSE;
	garr_stoermeldungen[st_config.i16_meld_startindex + 19] := FALSE;
	
	garr_betriebsmeldungen[st_config.i16_meld_startindex + 0] := FALSE;
	garr_betriebsmeldungen[st_config.i16_meld_startindex + 1] := FALSE;
	garr_betriebsmeldungen[st_config.i16_meld_startindex + 2] := FALSE;
	garr_betriebsmeldungen[st_config.i16_meld_startindex + 3] := FALSE;
	garr_betriebsmeldungen[st_config.i16_meld_startindex + 4] := FALSE;
	garr_betriebsmeldungen[st_config.i16_meld_startindex + 5] := FALSE;
	garr_betriebsmeldungen[st_config.i16_meld_startindex + 6] := FALSE;
	garr_betriebsmeldungen[st_config.i16_meld_startindex + 7] := FALSE;
	garr_betriebsmeldungen[st_config.i16_meld_startindex + 8] := FALSE;
	garr_betriebsmeldungen[st_config.i16_meld_startindex + 9] := FALSE;
	garr_betriebsmeldungen[st_config.i16_meld_startindex + 10] := FALSE;
	garr_betriebsmeldungen[st_config.i16_meld_startindex + 11] := FALSE;
	garr_betriebsmeldungen[st_config.i16_meld_startindex + 12] := FALSE;
	garr_betriebsmeldungen[st_config.i16_meld_startindex + 13] := FALSE;
	garr_betriebsmeldungen[st_config.i16_meld_startindex + 14] := FALSE;
	garr_betriebsmeldungen[st_config.i16_meld_startindex + 15] := FALSE;
	garr_betriebsmeldungen[st_config.i16_meld_startindex + 16] := FALSE;
	garr_betriebsmeldungen[st_config.i16_meld_startindex + 17] := FALSE;
	garr_betriebsmeldungen[st_config.i16_meld_startindex + 18] := FALSE;
	garr_betriebsmeldungen[st_config.i16_meld_startindex + 19] := FALSE;
END_IF
END_PROGRAM

(* POU Gemeinsamkeiten17xx/Achsen/ST_Z_Achse, ST *)
PROGRAM ST_Z_Achse
VAR_INPUT
	st_config_achse						: struct_ecd_config;
	st_ctrl_in								: struct_ctrl_in;
	e_steuerung_ein						: BOOL;
	e_ba_mit_bedingungen				: BOOL;
	e_tuere_vorne_offen					: BOOL;
	e_tuere_hinten_offen					: BOOL;

	b_start_in							: BOOL;
	lr_Achspos_in						: LREAL;
	lr_Velo_in							: LREAL;
	enu_cmd_in							: enum_ecd_cmd;
END_VAR
VAR_IN_OUT
	st_visu								: struct_ecd_visu;
END_VAR
VAR_OUTPUT
	st_ctrl_out							: struct_ctrl_out;
	t_Z_Achse_ausfahren				: TIME := t#0ms;
	t_Bestueckung					: TIME := t#0ms;
	t_Z_Achse_einfahren				: TIME := t#0ms;
	lr_RecPos						: LREAL;
END_VAR
VAR
	st_sm						 		: struct_ecd_meldungen;
	st_drive_cmd							: struct_ecd_cmd;
	st_drive_cmd_y_achse					: struct_ecd_cmd;
	fb_ton_wz							: TON;
	fb_ton_quitt							: TON;
	fb_ton_wz_disable						: TON;
	fb_ton_taktzeitmessung_wt_wechsel		: TON;
	fb_ton_taktzeitmessung_bestuecken		: TON;
	fb_r_trig_tippen						: R_TRIG;
	fb_f_trig_tippen						: F_TRIG;
	fb_r_trig_taste_plus					: R_TRIG;
	fb_r_trig_start							: R_TRIG;
	fb_r_trig_start_in						: R_TRIG;
	fb_r_trig_hand_dialog					: R_TRIG;
	fb_r_trig_nullpunkt_setzen				: R_TRIG;
	fb_axis								: ST_AxisJobCtrl_Motion;
	fb_axis_y_achse						: ST_AxisJobCtrl_Cam_Gear;
	fb_state_entry							: ST_StateEntry;
	fb_ton_uez							: TON;
	i									: DINT := 0;
	k									: DINT := 0;
	lr_pos_ohneverschiebung			: LREAL;
	fb_r_trig_limit_sensor_positiv			: R_TRIG;
	fb_r_trig_limit_sensor_negativ			: R_TRIG;
	fb_r_trig_skalierungsnocken				: R_TRIG;
	lr_slave_position						: LREAL := 0.0;
	i16_auftrag_cameditor					: enum_auftrag_cameditor;
	i16_kollisionszaehler					: INT := 0;
	b_hand_dialog_aktiv					: BOOL := FALSE;
	b_all_state_parts_ok					: BOOL := FALSE;
	b_kommt_von_init						: BOOL := FALSE;
	i32_UsedTool						: DINT := 0;

	sm_positionsueberwachung				: BOOL := FALSE;
	sm_werkzeugreihenfolge_nicht_io		: BOOL := FALSE;
	sm_keine_bandfreigabe				: BOOL := FALSE;
	sm_tagnummer_ungueltig				: BOOL := FALSE;
	sm_typ_bestueckprogramm_falsch	: BOOL := FALSE;
	sm_keine_rafo_im_einzug		: BOOL := FALSE;


	bm_kein_Pin_im_BB				: BOOL := FALSE;

	(* Kurvenscheibeneditor *)
	i16_startpunkt_mf_tab					: INT := 0;

	st_geschwindigkeiten					: struct_ecd_geschwindigkeiten;
	e_referenz_sensor						AT %I* : BOOL;
	i16_torque							AT %I* : INT;
	i16_DigitalInput						AT %I* : INT;

	lr_vmax_festo							: LREAL := 100.0;

	lr_ReduzierungOverride				: LREAL := 1.0;

	zeit_wt_wechsel						: DINT := 0;
	zeit_wt_bestuecken					: DINT := 0;

	fb_Z_Achse_einfahren			: ST_Taktzeit;
	fb_Bestueckung					: ST_Taktzeit;
	fb_Z_Achse_ausfahren	: ST_Taktzeit;

	lr_decceleration_nothalt				: LREAL;
	lr_decceleration_normal				: LREAL;

	i32_anzahl_rasterfolie				: DINT := 0;

	b_rastnase_vorhanden_vorne			: BOOL;
	b_rastnase_vorhanden_hinten			: BOOL;
	bm_rastnasen_1_fehlt					: BOOL;
	bm_rastnasen_2_fehlt					: BOOL;
	e_kontrolle_rastnase 			AT %I* : BOOL;
	b_teach_pruef_pos1					: BOOL;
	b_teach_pruef_pos2					: BOOL;

	i16_state_msg						: INT;
	Teile_nach_Bandwechsel				: BOOL;
	fb_r_trig_Bandwechsel					: R_TRIG;

	lr_MaxSoftPosLimit					:LREAL;
	lr_MinSoftPosLimit						:LREAL;
	b_EndlageErreicht						:BOOL;
	fb_r_trig_Endlage						: R_TRIG;
	i16_state_msg2						: INT;
END_VAR
(* Die Z-Achse ist der Masterablauf. Sie "weis" wann es losgeht und kennt das Bestückbild.
 * Die Z-Achse schaltet die Bestückachse als Master der Kurvenscheibe ein und startet diese. *)

(* Zeiten *)
fb_ton_wz(IN:= , PT:= , Q=>  , ET=> );
fb_ton_uez(IN:= , PT:= , Q=>  , ET=> );
fb_ton_quitt(IN:= , PT:= t#100ms, Q=> , ET=> );
fb_ton_wz_disable(IN:= , PT:= t#500ms, Q=> , ET=> );

fb_ton_taktzeitmessung_wt_wechsel(IN:= , PT:= t#2h, Q=> , ET=> );
fb_ton_taktzeitmessung_bestuecken(IN:= , PT:= t#2h, Q=> , ET=> );

(*Taktzeitmessung*)
fb_Z_Achse_einfahren(b_start:= , t_zeit=> );
fb_Bestueckung(b_start:= , t_zeit=> );
fb_Z_Achse_ausfahren(b_start:= , t_zeit=> );

(* Flanken *)
fb_r_trig_limit_sensor_positiv(CLK:= st_config_achse.b_limitsensor_positiv_vorhanden AND NOT fb_axis.e_limit_sensor_positive, Q=> );
fb_r_trig_limit_sensor_negativ(CLK:= st_config_achse.b_limitsensor_negativ_vorhanden AND NOT fb_axis.e_limit_sensor_negative, Q=> );
fb_r_trig_taste_plus(CLK:= ST_Euchner_Handbedienpult.b_Taste_Plus, Q=> );
fb_r_trig_start(CLK:= st_ctrl_in.b_start, Q=> );
fb_r_trig_start_in(CLK:= b_start_in, Q=> );
fb_r_trig_skalierungsnocken(CLK:= nockenschaltwerk_bestueckachse.fb.arr_spur[SP_START_SKALIERUNG], Q=> );
fb_r_trig_hand_dialog(CLK:= b_hand_dialog_aktiv, Q=> );
fb_r_trig_nullpunkt_setzen(CLK:=axis_z_achse.st_visu.b_nullpunkt_setzen);

(* Berechnung Override Reduzierung wenn Y-Achse die Rampe fahren muss *)
IF 	gst_datensatz.st_wkz.bFahreSofortAufUebergabePosition AND
	((z_achse.NcToPlc.ActPos > gst_datensatz.st_wkz.st_yz_tisch.r_wkz_einfahrpos_z - 20 AND
	gst_datensatz.st_wkz.b_variable_einfahrposition) OR
	(z_achse.NcToPlc.ActPos > ST_MotionFunctionPoints.YZTischMasterPos2 - 20 AND
	NOT gst_datensatz.st_wkz.b_variable_einfahrposition)) THEN
	lr_ReduzierungOverride := gst_datensatz.st_wkz.r_auto_z / st_geschwindigkeiten.lr_auto_max;
ELSE
	lr_ReduzierungOverride := 1;

END_IF


(*Meldung Teile nach Bandwechsel*)
fb_r_trig_Bandwechsel(CLK:= Teile_nach_Bandwechsel , Q=> );
IF fb_r_trig_Bandwechsel.Q  THEN
	i16_state_msg := 1;
END_IF

(*Produktionsmeldung für Übergabe zu lange*)
CASE i16_state_msg OF
	1: (*Warten bis keine ander Produktions Meldung ansteht *)
		IF	TestAndSet(ST_Message_Produktion.LockFlag) THEN
			ST_Message_Produktion.ClearMessageLines();
			i16_state_msg := 2;
		END_IF

	2:  (*Produktions Meldung*)
		Visu.MeldungProduktion.Color_R := 255;
		Visu.MeldungProduktion.Color_G := 255;
		Visu.MeldungProduktion.Color_B := 0;
		IF visu.s_akt_sprache = 'de' THEN
			Visu.MeldungProduktion.Name:=('Teile nach Bandwechsel');
		ELSIF visu.s_akt_sprache = 'en' THEN
			Visu.MeldungProduktion.Name:=('Teile nach Bandwechsel');
		ELSIF visu.s_akt_sprache = 'cz' THEN
			Visu.MeldungProduktion.Name:=('Teile nach Bandwechsel');
		END_IF
		Visu.MeldungProduktion.ShowMessage := TRUE;
		Visu.MeldungProduktion.Button1.sichtbar:=TRUE;	(*OK*)
		Visu.MeldungProduktion.Button1.Text:='Ok';
		i16_state_msg := 3;

	3:  (*Warte auf OK*)
		IF Visu.MeldungProduktion.Button1.tasten THEN
			i16_state_msg:=0;
		END_IF
END_CASE


(* Achse steuern *)
fb_axis(
	e_referenznocken:= ,
	b_refsensor_vorhanden:= st_config_achse.b_refsensor_vorhanden,
	b_limitsensor_positiv_vorhanden:= st_config_achse.b_limitsensor_positiv_vorhanden,
	b_limitsensor_negativ_vorhanden:= st_config_achse.b_limitsensor_negativ_vorhanden,
	i16_achstyp := st_config_achse.i16_achstyp,
	lr_override_vorgabe:= ST_TippTasten.lr_override * lr_ReduzierungOverride,
	st_position:= ,
	mc_richtung_modulo:= ,
	mc_richtung_velocity:= ,
	mc_referenzmodus:= ,
	mc_buffermode_axis:= ,
	ui16_soeparam_write_value:= ,
	w_idn:= ,
	i16_nc_parameter_nummer:= ,
	r_wert_nc_write_parameter:= ,
	st_vorgabe_geschwindigkeiten:= st_geschwindigkeiten,
	lr_soll_geschwindigkeit:= ,
	b_bedingung_sls:= NOT e_tuere_vorne_offen OR NOT e_tuere_hinten_offen,
	st_ads_info := ,
	st_eccoe_sdo := ,
	st_masterachse:= z_achse,
	st_visu_axis:= st_visu,
	st_ecd_cmd:= st_drive_cmd,
	ui16_soeparam_read_value=> ,
	r_wert_nc_read_parameter=> ,
	lr_RecPos=> lr_RecPos,
	b_TriggerInput:=i16_DigitalInput.1, (*1*)
	b_FallingEdge:=TRUE);

CASE gst_datensatz.st_md.i16_typ_zelle OF
	KEINE_ZELLE:
		;

	BESTUECKZELLE_1700:
		IF gi16_betriebsart = HAND THEN
			(* Bei manuellem Fahren der Slaveachse, muss diese erst entkoppelt werden *)
			IF ST_Y_Achse.b_hand_dialog_aktiv AND y_achse.NcToPlc.CoupleState > 0 THEN
				st_drive_cmd_y_achse.enu_cmd := CAM_OUT_SLAVE;
			END_IF
			(* Achse mit dem Euchner Handbediengerät vorwärts und rückwärts Bewegen*)
			IF fb_r_trig_hand_dialog.Q THEN
				IF y_achse.NcToPlc.CoupleState > 0 THEN
					st_drive_cmd_y_achse.enu_cmd := CAM_OUT_SLAVE;
				END_IF
				fb_state_entry.i16_next_step := HANDRAD;
			END_IF
		END_IF

		IF y_achse.NcToPlc.CoupleState > 0 OR st_drive_cmd_y_achse.enu_cmd > NO_COMMAND THEN
			(* Kurvenscheibenkopplung ein/ausschalten *)
			fb_axis_y_achse(
				r_getriebefaktor:= ,
				r_master_position:= ,
				mc_activation_mode_camin:= ,
				lr_activation_position_camin:= ,
				mc_activation_mode_scaleing:= ,
				lr_activation_position_scaleing:= ,
				mc_buffermode_axis:= ,
				mc_cam_table_id:= 2 ,
				mc_cam_point_id:= ,
				mc_motion_function_point:= ,
				st_camin_options:= ,
				st_camexchange_options:= ,
				mc_reference_cam_table_id:= ,
				st_camscaling_data:= ,
				st_masterachse:= z_achse,
				st_slaveachse:= y_achse,
				st_ecd_cmd:= st_drive_cmd_y_achse );
		END_IF

	BESTUECKZELLE_1720:
		IF gi16_betriebsart = HAND THEN
			(* Achse mit dem Euchner Handbediengerät vorwärts und rückwärts Bewegen*)
			IF fb_r_trig_hand_dialog.Q THEN
				fb_state_entry.i16_next_step := HANDRAD;
			END_IF
		END_IF

	RASTERFOLIE:
		IF gi16_betriebsart = HAND THEN
			(* Bei manuellem Fahren der Slaveachse, muss diese erst entkoppelt werden *)
			IF ST_Y_Achse.b_hand_dialog_aktiv AND y_achse.NcToPlc.CoupleState > 0 THEN
				st_drive_cmd_y_achse.enu_cmd := CAM_OUT_SLAVE;
			END_IF
			(* Achse mit dem Euchner Handbediengerät vorwärts und rückwärts Bewegen*)
			IF fb_r_trig_hand_dialog.Q THEN
				IF y_achse.NcToPlc.CoupleState = 3 THEN
					st_drive_cmd_y_achse.enu_cmd := CAM_OUT_SLAVE;
				END_IF
				fb_state_entry.i16_next_step := HANDRAD;
			END_IF
		END_IF

		IF y_achse.NcToPlc.CoupleState > 0 OR st_drive_cmd_y_achse.enu_cmd > NO_COMMAND THEN
			(* Kurvenscheibenkopplung ein/ausschalten *)
			fb_axis_y_achse(
				r_getriebefaktor:= ,
				r_master_position:= ,
				mc_activation_mode_camin:= ,
				lr_activation_position_camin:= ,
				mc_activation_mode_scaleing:= ,
				lr_activation_position_scaleing:= ,
				mc_buffermode_axis:= ,
				mc_cam_table_id:= 2 ,
				mc_cam_point_id:= ,
				mc_motion_function_point:= ,
				st_camin_options:= ,
				st_camexchange_options:= ,
				mc_reference_cam_table_id:= ,
				st_camscaling_data:= ,
				st_masterachse:= z_achse,
				st_slaveachse:= y_achse,
				st_ecd_cmd:= st_drive_cmd_y_achse );
		END_IF
END_CASE


IF gi16_betriebsart = HAND THEN
	(* Button in der Oberfläche zum setzen des Nullpunktes *)
	IF fb_r_trig_nullpunkt_setzen.Q THEN
		fb_state_entry.i16_next_step :=	NULLPUNKT_SETZEN;
	END_IF
END_IF

(*Meldung Achse hat Endlage überfahren*)
IF lr_MaxSoftPosLimit<>0 AND
  lr_MaxSoftPosLimit < gst_datensatz.st_md.st_md_z_achse.lr_wt_uebergabepos  THEN
	b_EndlageErreicht:= TRUE;
ELSE
	b_EndlageErreicht:=FALSE;
END_IF

fb_r_trig_Endlage(CLK:= b_EndlageErreicht , Q=> );

IF fb_r_trig_Endlage.Q THEN
	i16_state_msg2 := 1;
END_IF

(*Produktionsmeldung für Endlage überfahren*)
CASE i16_state_msg2 OF
	1: (*Warten bis keine ander Produktions Meldung ansteht *)
		IF	TestAndSet(ST_Message_Produktion.LockFlag) THEN
			ST_Message_Produktion.ClearMessageLines();
			i16_state_msg2 := 2;
		END_IF

	2:  (*Produktions Meldung*)
		Visu.MeldungProduktion.Color_R := 255;
		Visu.MeldungProduktion.Color_G := 255;
		Visu.MeldungProduktion.Color_B := 0;
		IF visu.s_akt_sprache = 'de' THEN
			Visu.MeldungProduktion.Name:='Z-Achse WT Übergabepos größer als Endlage';
		ELSIF visu.s_akt_sprache = 'en' THEN
			Visu.MeldungProduktion.Name:='Z-Achse WT Übergabepos größer als Endlage';
		ELSIF visu.s_akt_sprache = 'cz' THEN
			Visu.MeldungProduktion.Name:='Z-Achse WT Übergabepos größer als Endlage';
		END_IF
		Visu.MeldungProduktion.ShowMessage := TRUE;
		Visu.MeldungProduktion.Button1.sichtbar:=FALSE;	(*OK*)
		Visu.MeldungProduktion.Button1.Text:='Ok';
		i16_state_msg2 := 3;

	3:  (*Warte auf OK*)
		IF NOT b_EndlageErreicht THEN
			ST_Message_Produktion.b_PM_Quitt:=TRUE;
			i16_state_msg2:=0;
		END_IF
END_CASE


(* =======================================Toplevel========================================== *)
(* Starte Inbetriebnahme-Sequenz *)
IF st_ctrl_in.b_gehe_step_ibn THEN
	fb_state_entry.i16_next_step := INBETRIEBNAHME;
END_IF

(* =====Achse wird disabled===== *)
IF (NOT e_steuerung_ein OR NOT e_ba_mit_bedingungen) AND z_achse.Status.Operational THEN
	st_drive_cmd.enu_cmd := POWER_DISABLE;
END_IF

IF fb_state_entry.i16_next_step > INIT AND fb_state_entry.i16_next_step < FEHLER THEN
	(* =====Fehler vom Achskontroller===== *)
	IF st_drive_cmd.b_job_fehler OR st_drive_cmd_y_achse.b_job_fehler THEN
		fb_state_entry.i16_next_step := FEHLER;
	END_IF

	IF fb_state_entry.i16_next_step > 40 THEN
		(* Devicefehler *)
		IF z_achse.Status.Error THEN
			st_sm.b_achsfehler := TRUE;
			fb_state_entry.i16_next_step := FEHLER;
		ELSIF z_achse.Status.DriveDeviceError THEN
			st_sm.b_devicefehler := TRUE;
			fb_state_entry.i16_next_step := FEHLER;
		END_IF
	END_IF

	IF fb_state_entry.i16_next_step < STOP THEN
		(* =====Achse wird gestoppt===== *)
		IF st_ctrl_in.b_stop THEN
			fb_state_entry.i16_next_step := STOP;
		ELSIF fb_state_entry.i16_next_step < HALT THEN
			(* =====Achse wird angehalten===== *)
			IF st_ctrl_in.b_halt THEN
				fb_state_entry.i16_next_step := HALT;
			END_IF
		END_IF
	END_IF
END_IF

(* ======================================Schrittkette======================================== *)
fb_state_entry(
	i16_next_step:= , 
	i16_pos:= 1,
	s_debugtext:= ,
	E=> ,
	X=> ,
	i16_step=> ,
	i16_last_step=> );

CASE fb_state_entry.i16_step OF
(*=======================================================*)
	INIT_OBJ:
		IF st_config_achse.b_config_fertig THEN
			fb_state_entry.i16_next_step := 1;
		END_IF

(*=======================================================*)
	1:	(* Warte bis NetID´s der Slaves ausgelesen sind *)
		IF fb_state_entry.E THEN
			;
		END_IF

		(*-----------------------Weiterschaltbedingungen----------------------------*)
		IF ST_EthercatDiag.st_ctrl_out.b_fertig THEN
			fb_state_entry.i16_next_step := 2;
		END_IF

(*=======================================================*)
	2:	(* Spezifische NC-Achsparameter auslesen *)
		IF fb_state_entry.E THEN
			fb_axis.i16_nc_parameter_nummer := MaxVelocitySystem;
			st_drive_cmd.enu_cmd := READ_NC_PARAMETER;
		END_IF

		(*-----------------------Weiterschaltbedingungen----------------------------*)
		IF st_drive_cmd.enu_cmd = NO_COMMAND THEN
			lr_Velo_in:=st_geschwindigkeiten.lr_maximalgeschwindigkeit;
			st_geschwindigkeiten.lr_auto_max := st_geschwindigkeiten.lr_maximalgeschwindigkeit := fb_axis.r_wert_nc_read_parameter;
			st_geschwindigkeiten.lr_auto_min := 50;
			st_geschwindigkeiten.lr_jog := 100;
			fb_state_entry.i16_next_step := 3;
		END_IF

(*=======================================================*)
	3:	(* Spezifische NC-Achsparameter auslesen *)
		IF fb_state_entry.E THEN
			fb_axis.i16_nc_parameter_nummer := MaxAccelerationSystem;
			st_drive_cmd.enu_cmd := READ_NC_PARAMETER;
		END_IF

		(*-----------------------Weiterschaltbedingungen----------------------------*)
		IF st_drive_cmd.enu_cmd = NO_COMMAND THEN
			st_geschwindigkeiten.lr_beschleunigung := fb_axis.r_wert_nc_read_parameter;
			fb_state_entry.i16_next_step := 4;
		END_IF

(*=======================================================*)
	4:	(* Spezifische NC-Achsparameter auslesen *)
		IF fb_state_entry.E THEN
			fb_axis.i16_nc_parameter_nummer := MaxDecelerationSystem;
			st_drive_cmd.enu_cmd := READ_NC_PARAMETER;
		END_IF

		(*-----------------------Weiterschaltbedingungen----------------------------*)
		IF st_drive_cmd.enu_cmd = NO_COMMAND THEN
			st_geschwindigkeiten.lr_verzoegerung := fb_axis.r_wert_nc_read_parameter;
			lr_decceleration_normal := st_geschwindigkeiten.lr_verzoegerung;
			lr_decceleration_nothalt := 200000.0;
			fb_state_entry.i16_next_step := 5;
		END_IF

(*=======================================================*)
	5:	(* Spezifische NC-Achsparameter auslesen *)
		IF fb_state_entry.E THEN
			fb_axis.i16_nc_parameter_nummer := MaxJerk;
			st_drive_cmd.enu_cmd := READ_NC_PARAMETER;
		END_IF

		(*-----------------------Weiterschaltbedingungen----------------------------*)
		IF st_drive_cmd.enu_cmd = NO_COMMAND THEN
			st_geschwindigkeiten.lr_ruck := fb_axis.r_wert_nc_read_parameter;
			fb_state_entry.i16_next_step := 6;
		END_IF

(*=======================================================*)
	6:	(* Konfigurationen der Achse *)
		IF fb_state_entry.E THEN
			fb_axis.st_eccoe_sdo.s_ec_slave_net_id := ST_EthercatDiag.s_ec_slave_net_id[2];
			fb_axis.st_eccoe_sdo.ui16_slave_addr := st_config_achse.ui16_ethercat_adr;
		END_IF

		(*-----------------------Weiterschaltbedingungen----------------------------*)
		fb_state_entry.i16_next_step := 7;

(*=======================================================*)
	7:	(* Spezifische NC-Achsparameter auslesen *)
		IF fb_state_entry.E THEN
			fb_axis.i16_nc_parameter_nummer := AxisMinSoftPosLimit;
			st_drive_cmd.enu_cmd := READ_NC_PARAMETER;
		END_IF

		(*-----------------------Weiterschaltbedingungen----------------------------*)
		IF st_drive_cmd.enu_cmd = NO_COMMAND THEN
			lr_MinSoftPosLimit := fb_axis.r_wert_nc_read_parameter;
			fb_state_entry.i16_next_step := 8;
		END_IF


(*=======================================================*)
	8:	(* Spezifische NC-Achsparameter auslesen *)
		IF fb_state_entry.E THEN
			fb_axis.i16_nc_parameter_nummer := AxisMaxSoftPosLimit;
			st_drive_cmd.enu_cmd := READ_NC_PARAMETER;
		END_IF

		(*-----------------------Weiterschaltbedingungen----------------------------*)
		IF st_drive_cmd.enu_cmd = NO_COMMAND THEN
			lr_MaxSoftPosLimit := fb_axis.r_wert_nc_read_parameter;
			fb_state_entry.i16_next_step := FEHLER; (*in Fehler gehen damit die Achsen resetet werden. Sonst steigen die Achsen bei einem TC Restart aus*)
		END_IF

(*=======================================================*)
	INIT:
		IF fb_state_entry.E THEN
			fb_ton_wz.IN := FALSE;
			fb_ton_uez.IN	:= FALSE;
			fb_ton_quitt.IN := FALSE;
			fb_ton_taktzeitmessung_wt_wechsel.IN := FALSE;
			fb_ton_taktzeitmessung_bestuecken.IN := FALSE;
			b_start_in:=FALSE;
			st_ctrl_in.b_start:=FALSE;
			st_ctrl_out.b_busy:=FALSE;
			st_ctrl_out.b_fehler := FALSE;
			st_ctrl_out.b_fertig := FALSE;
			st_ctrl_out.b_fertig_2 := FALSE;
			st_ctrl_out.b_bereit := FALSE;
			st_ctrl_out.b_gestoppt := FALSE;
			st_ctrl_out.b_prebereit := FALSE;
			axis_y_achse.st_ctrl.in.b_start := FALSE;
			i16_kollisionszaehler := 0;
			(* Reset Stoermeldungen *)
			st_sm.b_achse_nicht_auf_startpos := FALSE;
			st_sm.b_achsfehler := FALSE;
			st_sm.b_devicefehler := FALSE;
			st_sm.b_keine_verfahrfreigabe := FALSE;
			st_sm.b_ende_skalierungs_nocke := FALSE;
			st_sm.b_ende_camming_nocke := FALSE;
			st_sm.b_skalierung_noch_aktiv := FALSE;
			sm_positionsueberwachung := FALSE;
			sm_werkzeugreihenfolge_nicht_io := FALSE;
			sm_keine_bandfreigabe := FALSE;
			sm_tagnummer_ungueltig := FALSE;
			sm_typ_bestueckprogramm_falsch := FALSE;
			sm_keine_rafo_im_einzug:=FALSE;

			bm_rastnasen_1_fehlt := FALSE;
			bm_rastnasen_2_fehlt := FALSE;

			bm_kein_Pin_im_BB:= FALSE;

			axis_y_achse.st_ctrl.in.b_start := FALSE;
			axis_y_achse.st_ctrl.in.b_start_2 := FALSE;
			axis_virt_master.st_ctrl.in.b_start := FALSE;
			rasterfolienmontage.st_ctrl.in.b_start := FALSE;
			balluff_tag_reader.st_ctrl.in.b_start_lesen := FALSE;
			balluff_tag_reader.st_ctrl.in.b_start_schreiben := FALSE;

			b_kommt_von_init := TRUE;

			fb_axis.mc_buffermode_axis := MC_Aborting;

			fb_axis.lr_soll_geschwindigkeit := gst_datensatz.st_wkz.r_auto_z;

			st_geschwindigkeiten.lr_verzoegerung := lr_decceleration_normal;
		END_IF

		IF y_achse.NcToPlc.CoupleState > 0 THEN
			st_drive_cmd_y_achse.enu_cmd := CAM_OUT_SLAVE;
		END_IF

		(*-----------------------Weiterschaltbedingungen----------------------------*)
		IF st_ctrl_in.b_preinit THEN
			fb_state_entry.i16_next_step := 15;
		END_IF

(*=======================================================*)
	15:	(* Reglerfreigabe wegnehmen *)
		IF fb_state_entry.E THEN
			st_drive_cmd.enu_cmd := POWER_DISABLE;
		END_IF

		(*-----------------------Weiterschaltbedingungen----------------------------*)
		IF st_drive_cmd.enu_cmd = NO_COMMAND THEN
			fb_state_entry.i16_next_step := 20;
		END_IF

(*=======================================================*)
	20:	(* Überprüfe Nullpunktverschiebung des Absolutwertgebers auf Korrektheit *)
		IF fb_state_entry.E THEN
			fb_axis.i16_nc_parameter_nummer := AxisEncoderOffset;	(* vom Datentyp MC_AxisParameter *)
			st_drive_cmd.enu_cmd := READ_NC_PARAMETER;
		END_IF

		(*-----------------------Weiterschaltbedingungen----------------------------*)
		IF st_drive_cmd.enu_cmd = NO_COMMAND THEN
			IF fb_axis.r_wert_nc_read_parameter = gst_datensatz.st_md.st_md_z_achse.lr_nullpunktverschiebung THEN
				CASE gst_datensatz.st_md.i16_typ_zelle OF
					KEINE_ZELLE:
						;

					BESTUECKZELLE_1700, RASTERFOLIE:
						fb_state_entry.i16_next_step := 35;
	
					BESTUECKZELLE_1720:
						fb_state_entry.i16_next_step := 40;
				END_CASE
			ELSE
				fb_state_entry.i16_next_step := 25;	(* Nullpunktverschiebung schreiben *)
			END_IF
		END_IF

(*=======================================================*)
	25:	(* Nullpunktverschiebung hat sich geändert, deshalb erst Null reinschreiben, um keinen Additionsfehler zu machen, *)
		(* weil der Wert der Verschiebung beim Neustart komplett auf die Achse geschrieben wird *)
		IF fb_state_entry.E THEN
			fb_axis.i16_nc_parameter_nummer := AxisEncoderOffset;
			fb_axis.r_wert_nc_write_parameter := 0.0;
			st_drive_cmd.enu_cmd := WRITE_NC_PARAMETER;
		END_IF

		(*-----------------------Weiterschaltbedingungen----------------------------*)
		IF st_drive_cmd.enu_cmd = NO_COMMAND THEN
			fb_state_entry.i16_next_step := 30;
		END_IF

(*=======================================================*)
	30:	(* Aktuelle Nullpunktverschiebung des Absolutwertgebers an die Achse senden *)
		IF fb_state_entry.E THEN
			fb_axis.i16_nc_parameter_nummer := AxisEncoderOffset;
			fb_axis.r_wert_nc_write_parameter := gst_datensatz.st_md.st_md_z_achse.lr_nullpunktverschiebung;
			st_drive_cmd.enu_cmd := WRITE_NC_PARAMETER;
		END_IF

		(*-----------------------Weiterschaltbedingungen----------------------------*)
		IF st_drive_cmd.enu_cmd = NO_COMMAND THEN
			CASE gst_datensatz.st_md.i16_typ_zelle OF
				KEINE_ZELLE:
					;

				BESTUECKZELLE_1700, RASTERFOLIE:
					fb_state_entry.i16_next_step := 35;

				BESTUECKZELLE_1720:
					fb_state_entry.i16_next_step := 40;
			END_CASE
		END_IF

(*=======================================================*)
	35:	(* CAM OUT Y-Achse *)
		IF fb_state_entry.E THEN
			st_drive_cmd_y_achse.enu_cmd := CAM_OUT_SLAVE;
		END_IF

		(*-----------------------Weiterschaltbedingungen----------------------------*)
		IF st_drive_cmd_y_achse.enu_cmd = NO_COMMAND AND NOT fb_state_entry.E THEN
			fb_state_entry.i16_next_step := 40;
		END_IF

(*=======================================================*)
	40:	(* Reglerfreigabe setzen , Reset wird bei Bedarf automatisch ausgeführt*)
		IF fb_state_entry.E THEN
			st_drive_cmd.enu_cmd := POWER_ENABLE;
		END_IF

		(*-----------------------Weiterschaltbedingungen----------------------------*)
		IF st_drive_cmd.enu_cmd = NO_COMMAND THEN
			fb_state_entry.i16_next_step := 50;
		END_IF

(*=======================================================*)
	50:	(* Nullpunktverschiebung ist geschrieben *)
		IF fb_state_entry.E THEN
			st_ctrl_out.b_prebereit := TRUE;
		END_IF

		(*-----------------------Weiterschaltbedingungen----------------------------*)
		IF st_ctrl_in.b_init THEN
			CASE gst_datensatz.st_md.i16_typ_zelle OF
				KEINE_ZELLE:
					;

				BESTUECKZELLE_1700, RASTERFOLIE:
					fb_state_entry.i16_next_step := 60;

				BESTUECKZELLE_1720:
					fb_state_entry.i16_next_step := 95;
			END_CASE
		END_IF

(*=======================================================*)
	60: (* Abfrage der Positionen von Z-Achse und Y-Achse *)

		(*-----------------------Weiterschaltbedingungen----------------------------*)
		IF 	z_achse.NcToPlc.ActPos > ST_MotionFunctionPoints.YZTischMasterPos3 AND
			ABS(y_achse.NcToPlc.ActPos - gst_datensatz.st_md.st_md_y_achse.lr_wt_uebergabepos) > 0.5
			THEN
				(* Y-Achse steht in Kollision mit Antriebskonus des Förderbands *)
				fb_state_entry.i16_next_step := 70;
		ELSE
			i16_kollisionszaehler := 0;
			fb_state_entry.i16_next_step := 80;
		END_IF

(*=======================================================*)
	70: (* Im Wiederhohlungsfall -> Fehler *)
		IF fb_state_entry.E THEN
			i16_kollisionszaehler := i16_kollisionszaehler + 1;
		END_IF

		(*-----------------------Weiterschaltbedingungen----------------------------*)
		IF i16_kollisionszaehler > 1 THEN
			sm_positionsueberwachung := TRUE;
			fb_state_entry.i16_next_step := FEHLER;
		ELSE
			fb_state_entry.i16_next_step := 75;
		END_IF

(*=======================================================*)
	75:	(* Fahre Z-Achse und damit Y-Achse aus der Kollisionsposition *)
		IF fb_state_entry.E THEN
			fb_axis.lr_soll_geschwindigkeit := gst_datensatz.st_wkz.r_auto_z;
			fb_axis.st_position.r_soll := ST_MotionFunctionPoints.YZTischMasterPos3;
			st_drive_cmd.enu_cmd := MOVE_ABSOLUTE;
		END_IF

		(*-----------------------Weiterschaltbedingungen----------------------------*)
		IF st_drive_cmd.enu_cmd = NO_COMMAND THEN
			fb_state_entry.i16_next_step := 80;
		END_IF

(*=======================================================*)
	80: (* Auslesen der Y-Position an der aktuellen Z-Position in der Kurvenscheibe *)
		IF fb_state_entry.E THEN
			fb_axis_y_achse.r_master_position := z_achse.NcToPlc.ActPos;
			st_drive_cmd_y_achse.enu_cmd := READ_SLAVE_DYNAMICS;
		END_IF

		(*-----------------------Weiterschaltbedingungen----------------------------*)
		IF st_drive_cmd_y_achse.enu_cmd = NO_COMMAND AND NOT fb_state_entry.E THEN
			fb_state_entry.i16_next_step := 85;
		END_IF

(*=======================================================*)
	85: (* Starte Y-Achse auf die entsprechende Position in der Kurvenscheibe *)
		IF fb_state_entry.E THEN
			lr_slave_position := fb_axis_y_achse.mc_read_camtable_slave_dynamics.SlavePosition;
			axis_y_achse.st_ctrl.in.b_start := TRUE;
		END_IF

		(*-----------------------Weiterschaltbedingungen----------------------------*)
		IF axis_y_achse.st_ctrl.out.b_fertig AND NOT fb_state_entry.E THEN
			axis_y_achse.st_ctrl.in.b_start := FALSE;
			fb_state_entry.i16_next_step := 90;
		END_IF

(*=======================================================*)
	90:	(* CAM IN Y-Achse *)
		IF fb_state_entry.E THEN
			fb_axis_y_achse.st_camscaling_data.SlaveScaling := 1;
			st_drive_cmd_y_achse.enu_cmd := CAM_IN_SLAVE;
		END_IF

		IF y_achse.NcToPlc.CoupleState = 0 THEN
			st_drive_cmd_y_achse.enu_cmd := CAM_IN_SLAVE;
		END_IF

		(*-----------------------Weiterschaltbedingungen----------------------------*)
		IF st_drive_cmd_y_achse.enu_cmd = NO_COMMAND AND NOT fb_state_entry.E THEN
			fb_state_entry.i16_next_step := 95;
		END_IF

(*=======================================================*)
	95:	(* Fahre Z-Achse auf die WT-Übergabeposition *)
		IF fb_state_entry.E THEN
			fb_axis.lr_soll_geschwindigkeit := gst_datensatz.st_wkz.r_auto_z;
			fb_axis.st_position.r_soll := gst_datensatz.st_md.st_md_z_achse.lr_wt_uebergabepos;
			st_drive_cmd.enu_cmd := MOVE_ABSOLUTE;
		END_IF

		(*-----------------------Weiterschaltbedingungen----------------------------*)
		IF st_drive_cmd.enu_cmd = NO_COMMAND THEN
			fb_state_entry.i16_next_step := BEREIT;
		END_IF

(*=======================================================*)
	BEREIT:
		IF fb_state_entry.E THEN
			st_ctrl_out.b_busy:=FALSE;
			st_ctrl_out.b_bereit := TRUE;
			st_ctrl_out.b_fertig := TRUE;
			bm_rastnasen_1_fehlt := FALSE;
			bm_rastnasen_2_fehlt := FALSE;
			enu_cmd_in:=NO_COMMAND;
		END_IF

		IF NOT gst_datensatz.st_wkz.b_rafo_auto_einf_aktiv THEN
			IF 	gst_datensatz.st_md.i16_typ_zelle = RASTERFOLIE AND
				NOT ST_Rasterfolieneinzug.fb_tof_gls_rafo_ende.Q THEN
				fb_state_entry.i16_next_step := FEHLER;
				sm_keine_rafo_im_einzug:=TRUE;
			END_IF
		END_IF

		(*-----------------------Weiterschaltbedingungen----------------------------*)
		IF fb_r_trig_start.Q  THEN
(*			(* Stoppe WT Wechselzeit *)
			zeit_wt_wechsel := TIME_TO_DWORD(fb_ton_taktzeitmessung_wt_wechsel.ET);
			fb_ton_taktzeitmessung_wt_wechsel.IN := FALSE;
			(* Starte Bestückzeit *)
			fb_ton_taktzeitmessung_bestuecken.IN := TRUE;*)
			fb_Z_Achse_einfahren(b_start:= TRUE, t_zeit=> );
			st_ctrl_out.b_fertig := FALSE;
			st_ctrl_out.b_busy:=TRUE;
			i32_anzahl_rasterfolie:=0;
			fb_state_entry.i16_next_step := 110;
		END_IF

		IF 	fb_r_trig_start_in.Q THEN		(*neu! zum Starten einer Positionierung von einem externen Prg.*)
			st_ctrl_out.b_fertig := FALSE;
			st_ctrl_out.b_busy:=TRUE;
			fb_state_entry.i16_next_step := 102;
		END_IF

(*=======================================================*)
	102:	(*Y Achse abkoppeln*)
		IF 	fb_state_entry.E THEN
			b_start_in:=FALSE;
		END_IF

		IF 	y_achse.NcToPlc.CoupleState > 0 THEN
			st_drive_cmd_y_achse.enu_cmd := CAM_OUT_SLAVE;
		ELSE
			fb_state_entry.i16_next_step := 103;
		END_IF

(*=======================================================*)
	103:
		(*-----------------------Weiterschaltbedingungen----------------------------*)
		IF	enu_cmd_in = NO_COMMAND THEN
			fb_state_entry.i16_next_step := BEREIT;
		ELSIF
			enu_cmd_in = CAM_IN_SLAVE THEN
			fb_state_entry.i16_next_step := 90;		 (* Y Achse Cam In und auf Grundstellung fahren   *)

		ELSE
			fb_state_entry.i16_next_step := 104;
		END_IF

(*=======================================================*)
	104: (* Positioniere Achse  *)
		IF 	fb_state_entry.E THEN
			fb_axis.st_position.r_soll := lr_Achspos_in ;
			fb_axis.lr_soll_geschwindigkeit:=lr_Velo_in;
			st_drive_cmd.enu_cmd := enu_cmd_in;
		END_IF

		(*-----------------------Weiterschaltbedingungen----------------------------*)
		IF 	st_drive_cmd.enu_cmd = NO_COMMAND THEN
			fb_state_entry.i16_next_step := BEREIT;
		END_IF

(*=======================================================*)
	110: (* WT-Tag mit RFID-Lesegerät auslesen *)
		IF fb_state_entry.E THEN
			balluff_tag_reader.st_ctrl.in.b_start_lesen := TRUE;
			balluff_tag_reader.fb.i16_addresse := 0;
			balluff_tag_reader.fb.i16_anzahl_byte := SIZEOF(gst_tag_data);
		END_IF

		(*-----------------------Weiterschaltbedingungen----------------------------*)
		IF balluff_tag_reader.st_ctrl.out.b_fertig AND NOT fb_state_entry.E THEN
			ST_Konvertiere_gelese_TagData();

			IF gst_tag_data.WpcNumber >= 1 AND gst_tag_data.WpcNumber <=50 THEN
				fb_state_entry.i16_next_step := 120;
			ELSE
				(* Fehler: Tagnummer ist nicht im gültigem Bereich *)
				sm_tagnummer_ungueltig := TRUE;
				fb_state_entry.i16_next_step := FEHLER;
			END_IF
		END_IF

		IF fb_state_entry.X THEN
			balluff_tag_reader.st_ctrl.in.b_start_lesen := FALSE;
			fb_ton_wz.IN := FALSE;
		END_IF

(*=======================================================*)
	120: (* Die WPCDaten vom ausgelesenen Tag abfragen *)
		IF fb_state_entry.E THEN
			CASE gst_datensatz.st_md.i16_typ_zelle OF
				KEINE_ZELLE:
					;
	
				BESTUECKZELLE_1700, RASTERFOLIE:
					(* Daten Gültig *)
					IF 	(gst_tag_data.StateParts[0] = PART_NEW OR gst_tag_data.StateParts[0] = PART_OK) OR
						hublift_links.st_config.b_station_aktiv OR visu.b_inbetriebnahme OR NOT gst_datensatz.st_md.b_wt_transport_aktiv
						THEN
							fb_state_entry.i16_next_step := 130;
					ELSE
						(* Einfach durchschleusen: Wir muessen nicht bearbeiten. z.B. für gst_tag_data.State01 = PART_DUMMY *)
						fb_state_entry.i16_next_step := BEREIT;
					END_IF

				BESTUECKZELLE_1720:
					(* Daten Gültig *)
					IF 	(gst_tag_data.StateParts[0] = PART_NEW AND gst_tag_data.StateParts[1] = PART_NEW) OR
						(gst_tag_data.StateParts[0] = PART_OK AND gst_tag_data.StateParts[1] = PART_OK) OR
						hublift_links.st_config.b_station_aktiv OR visu.b_inbetriebnahme OR NOT gst_datensatz.st_md.b_wt_transport_aktiv
						THEN
							fb_state_entry.i16_next_step := 130;
					ELSE
						(* Einfach durchschleusen: Wir muessen nicht bearbeiten *)
						fb_state_entry.i16_next_step := BEREIT;
					END_IF
			END_CASE
		END_IF

(*=======================================================*)
		130:	(* Prüfe Bandfreigabe *)

		(*-----------------------Weiterschaltbedingungen----------------------------*)
		CASE gst_datensatz.st_md.i16_typ_zelle OF
			KEINE_ZELLE:
				;

			BESTUECKZELLE_1700:
				IF 	zyl_bawe_querschub.fb.e_sensor1_eingefahren AND
					((gst_barcode_daten.b_band_links_ok AND gst_barcode_daten.b_band_ID_links_ok) OR
					ST_Virtuelle_Masterachse.b_merker_bandende_links) THEN
					fb_state_entry.i16_next_step := 140;
				ELSIF
					zyl_bawe_querschub.fb.e_sensor1_ausgefahren AND
					((gst_barcode_daten.b_band_rechts_ok AND gst_barcode_daten.b_band_ID_rechts_ok) OR
					ST_Virtuelle_Masterachse.b_merker_bandende_rechts) THEN
					fb_state_entry.i16_next_step := 140;
				ELSE
					sm_keine_bandfreigabe := TRUE;
					fb_state_entry.i16_next_step := 180; 	(*Plle mit NOK beschreiben danach FEHLER*)
				END_IF

			BESTUECKZELLE_1720:
				IF 	(gst_barcode_daten.b_band_ok AND gst_barcode_daten.b_band_ID_links_ok AND gst_barcode_daten.b_band_ID_rechts_ok)  OR
					ST_Virtuelle_Masterachse.b_merker_bandende_rechts OR
					ST_Virtuelle_Masterachse.b_merker_bandende_links THEN
					fb_state_entry.i16_next_step := 140;

				ELSE
					sm_keine_bandfreigabe := TRUE;
					fb_state_entry.i16_next_step := 180; 	(*Plle mit NOK beschreiben danach FEHLER*)
				END_IF

			RASTERFOLIE:
				IF 	gst_barcode_daten.b_band_links_ok THEN
					fb_state_entry.i16_next_step := 140;

				ELSE
					sm_keine_bandfreigabe := TRUE;
					fb_state_entry.i16_next_step := 180; 	(*Plle mit NOK beschreiben danach FEHLER*)
				END_IF

		END_CASE

(*=======================================================*)
	140:	(* Muss das Bestückbild neu von Tag ausgelesen werden? *)


		(*-----------------------Weiterschaltbedingungen----------------------------*)
		IF 	s_alte_artikelnummer = gst_datensatz.st_md.s_aktuelle_artikelnummer AND
			gst_datensatz.st_md.b_wt_transport_aktiv AND
			NOT b_kommt_von_init THEN
			fb_state_entry.i16_next_step := 160;
		ELSE
			fb_state_entry.i16_next_step := 150;
		END_IF

(*=======================================================*)
	150:	(* Bestückbild aus DB von Festplatte einlesen. *)
		IF fb_state_entry.E THEN
			b_kommt_von_init := FALSE;
			gi16_bbgen_auftrag := LESE_BESTUECKBILD; (*und ISK*)
		END_IF

		(*-----------------------Weiterschaltbedingungen----------------------------*)
		IF 	gi16_bbgen_auftrag = KEIN_BB_AUFTRAG THEN
			s_alte_artikelnummer := gst_datensatz.st_md.s_aktuelle_artikelnummer;
			fb_state_entry.i16_next_step := 160;
		END_IF

(*=======================================================*)
	160:	(* Suche nach "Pruef" in Artikelnummer (nur für Rasterfolie) *)

		(*-----------------------Weiterschaltbedingungen----------------------------*)
		CASE gst_datensatz.st_md.i16_typ_zelle OF

			BESTUECKZELLE_1700, BESTUECKZELLE_1720:
				fb_state_entry.i16_next_step := 170;

			RASTERFOLIE:
				IF 	(FIND(gst_datensatz.st_md.s_aktuelle_artikelnummer, 'ruef') > 0 OR			(*es wird nur auf ruef abgefragt, weil das P groß oder klein sein kann*)
					FIND(gst_datensatz.st_md.s_aktuelle_artikelnummer,'erth') > 0)THEN
					fb_state_entry.i16_next_step := 370;	(* nicht Bestücken *)
				ELSE
					fb_state_entry.i16_next_step := 170;
				END_IF

		END_CASE

(*=======================================================*)
	170: (* Prüfe Werkzeugreihenfolge *)
		(* 	3 Fälle:
			1:	- PART_NEW	--->	Wir sind die erste Station
			2:	- PART_OK	--->	Vorgänger hat Station Ok bearbeitet
				-			--->	Prüfe dass diese LastUsedTool in der Liste vor unserer Station steht

			3:	- PART_NOK	-->	Kommt hier gar nicht an, trotzdem Fehler abfangen
				- PART_NO	-->	Kommt hier gar nicht an, trotzdem Fehler abfangen
		*)	
		IF fb_state_entry.E THEN
			CASE gst_datensatz.st_md.i16_typ_zelle OF
				KEINE_ZELLE:
					;

				BESTUECKZELLE_1700, BESTUECKZELLE_1720, RASTERFOLIE:
					IF gst_datensatz.st_md.i16_typ_bestueckmodus<>BESTUECKUNG_MANUAL  AND gst_datensatz.st_md.b_wt_transport_aktiv THEN

						i32_UsedTool:=-1;
						k:=-1;
						FOR k := 0 TO 4 DO      (*Werkzeuggruppen durchsuchen*)
							i:=-1;

							CASE gst_datensatz.st_md.i16_typ_bestueckmodus OF

								BESTUECKUNG_MANUAL:
											;
								BESTUECKUNG_HALBAUTO:

									FOR i := 0 TO MaxNoOfWkz DO
										IF 	gst_bestueckbild_halbauto.s_wkzgruppe[k].s_wkznummer[i] = gst_datensatz.st_md.s_aktuelles_wkz THEN
											i32_UsedTool:=i;
										END_IF
									END_FOR

								BESTUECKUNG_AUTO:

									FOR i := 0 TO MaxNoOfWkz DO
										IF 	gst_bestueckbild.s_wkzgruppe[k].s_wkznummer[i] = gst_datensatz.st_md.s_aktuelles_wkz THEN
											i32_UsedTool:=i;
										END_IF
									END_FOR

								ELSE
									sm_typ_bestueckprogramm_falsch := TRUE;
									fb_state_entry.i16_next_step := FEHLER;
							END_CASE

						END_FOR

						(* ------- Fall 1-------- *)
						IF gst_tag_data.StateParts[0]= PART_NEW THEN
							IF 	i32_UsedTool<>-1 THEN
								gst_tag_data.LastUsedTool := DINT_TO_BYTE(i32_UsedTool);
								fb_state_entry.i16_next_step := 190;
							ELSE
							(* NOk *)
								sm_werkzeugreihenfolge_nicht_io := TRUE;
								fb_state_entry.i16_next_step := 180; 	(*Pille mit NOK beschreiben danach FEHLER*)
							END_IF

						(* ------- Fall 2-------- *)
						ELSIF gst_tag_data.StateParts[0] = PART_OK THEN

							(* Ok *)
							IF 	i32_UsedTool<>-1 AND
							 	gst_tag_data.LastUsedTool < i32_UsedTool AND
								i32_UsedTool < gst_tag_data.LastUsedTool+3 THEN
								gst_tag_data.LastUsedTool := DINT_TO_BYTE(i32_UsedTool);
								fb_state_entry.i16_next_step := 190;
							ELSIF gst_tag_data.LastUsedTool = i32_UsedTool THEN
								fb_state_entry.i16_next_step := BEREIT;	(* nichts tun, ich habe schon bestückt *)
							ELSE
							(* NOk *)
								sm_werkzeugreihenfolge_nicht_io := TRUE;
								fb_state_entry.i16_next_step := 180; 	(*Pille mit NOK beschreiben danach FEHLER*)
							END_IF
						(* ------- Fall 3-------- *)
						ELSE
							sm_werkzeugreihenfolge_nicht_io := TRUE;
							fb_state_entry.i16_next_step := 180; 	(*Pille mit NOK beschreiben danach FEHLER*)
						END_IF
					ELSE
						(* Manuelle BB Anwahl *)
						gst_tag_data.LastUsedTool := 0;
						fb_state_entry.i16_next_step := 190;
					END_IF
			END_CASE
		END_IF

(*=======================================================*)
	180: (* Markiere WT als schlecht, weil Werkzeugreihenfolge nicht passt und Ende mit Fehler. *)
		IF fb_state_entry.E THEN
			ST_Markiere_WT_NIO();
		END_IF

		(*-----------------------Weiterschaltbedingungen----------------------------*)
		IF balluff_tag_reader.st_ctrl.out.b_fertig AND NOT fb_state_entry.E THEN
			(* Ok: Daten wurden auf die Pille geschrieben *)
			balluff_tag_reader.st_ctrl.in.b_start_schreiben := FALSE;
			fb_state_entry.i16_next_step := FEHLER;
		END_IF

(*=======================================================*)
	190:	(* Werkzeugreihenfolge in Ordnung *)

		(*-----------------------Weiterschaltbedingungen----------------------------*)
		CASE gst_datensatz.st_md.i16_typ_zelle OF
			KEINE_ZELLE:
				;

			BESTUECKZELLE_1700, RASTERFOLIE:
				IF 	gst_PersDaten.b_Zelle_nicht_in_Betrieb AND (FIND(gst_datensatz.st_md.s_aktuelle_artikelnummer,'ruef') = 0 AND			(*es wird nur auf ruef abgefragt, weil das P groß oder klein sein kann*)
					FIND(gst_datensatz.st_md.s_aktuelle_artikelnummer,'erth') = 0) THEN
					fb_state_entry.i16_next_step := 195;
				ELSE
					IF 	gst_datensatz.st_md.b_tagreader_fahrend THEN
						fb_state_entry.i16_next_step := 200;
					ELSE
						fb_state_entry.i16_next_step := 210;
					END_IF
				END_IF


				(*Abbruch wenn kein Pin bestückt wird*)
				IF	gst_datensatz.st_bestueckprogramm.i32_anzahl=0 THEN
					fb_state_entry.i16_next_step := 350;
					bm_kein_Pin_im_BB:= TRUE;
					IF FIND(gst_datensatz.st_md.s_aktuelle_artikelnummer,'ruef') = 0 AND			(*es wird nur auf ruef abgefragt, weil das P groß oder klein sein kann*)
						FIND(gst_datensatz.st_md.s_aktuelle_artikelnummer,'erth') = 0THEN
						gst_PersDaten.b_Zelle_nicht_in_Betrieb := TRUE;
					END_IF
				ELSE
					bm_kein_Pin_im_BB:= FALSE;
				END_IF

			BESTUECKZELLE_1720:
				IF 	gst_PersDaten.b_Zelle_nicht_in_Betrieb AND (FIND(gst_datensatz.st_md.s_aktuelle_artikelnummer,'ruef') = 0 AND			(*es wird nur auf ruef abgefragt, weil das P groß oder klein sein kann*)
					FIND(gst_datensatz.st_md.s_aktuelle_artikelnummer,'erth') = 0) THEN
					fb_state_entry.i16_next_step := 395;
				ELSE
					IF gst_datensatz.st_md.	b_tagreader_fahrend THEN
						fb_state_entry.i16_next_step := 400;
					ELSE
						fb_state_entry.i16_next_step := 405;
					END_IF
				END_IF

				(*Abbruch wenn kein Pin bestückt wird*)
				IF	gst_datensatz.st_bestueckprogramm.i32_anzahl=0 THEN
					fb_state_entry.i16_next_step := 460;
					bm_kein_Pin_im_BB:= TRUE;
					IF 	FIND(gst_datensatz.st_md.s_aktuelle_artikelnummer,'ruef') = 0 AND			(*es wird nur auf ruef abgefragt, weil das P groß oder klein sein kann*)
						FIND(gst_datensatz.st_md.s_aktuelle_artikelnummer,'erth') = 0 THEN
						gst_PersDaten.b_Zelle_nicht_in_Betrieb := TRUE;
					END_IF
				ELSE
					bm_kein_Pin_im_BB:= FALSE;
				END_IF
		END_CASE

(*=======================================================*)
	195: (*Warten bis keine ander Produktions Meldung ansteht *)
		IF	TestAndSet(ST_Message_Produktion.LockFlag) THEN
			ST_Message_Produktion.ClearMessageLines();
			fb_state_entry.i16_next_step := 196;
		END_IF

(*=======================================================*)
	196:  (*Produktions Meldung*)
		Visu.MeldungProduktion.Color_R := 255;
		Visu.MeldungProduktion.Color_G := 0;
		Visu.MeldungProduktion.Color_B := 0;
		IF visu.s_akt_sprache = 'de' THEN
			Visu.MeldungProduktion.Name:='Zelle war nicht in Betrieb, bitte Instandhalter informieren!$R$N$R$NÖler,Bestückposition, Seitenversatz und Biegewinkel kontrollieren$R$NMeldung kann nur eingeloggt quittiert werden';
		ELSIF visu.s_akt_sprache = 'en' THEN
			Visu.MeldungProduktion.Name:='Station has not been used for last order, please inform Maintenance Technician!$R$N$R$Ncheck oiler, stich position, left/right and bending angle$R$Nmessage can only be acknowledged when logged in';
		ELSIF visu.s_akt_sprache = 'cz' THEN
			Visu.MeldungProduktion.Name:='Bunka nebyla v provozu, informujte prosim serizovace. Zkontrolujte olej, nastaveni os a uhel ohybu.$R$NZprávu lze potvrdit jen po prihlaseni ';
		END_IF
		Visu.MeldungProduktion.ShowMessage := TRUE;
		Visu.MeldungProduktion.Button1.sichtbar:=TRUE;	(*OK*)
		Visu.MeldungProduktion.Button1.Text:='Ok';

		(*-----------------------Weiterschaltbedingungen----------------------------*)
		IF visu.b_logon THEN
			IF Visu.MeldungProduktion.Button1.tasten THEN
				IF gst_datensatz.st_md.	b_tagreader_fahrend THEN
					fb_state_entry.i16_next_step := 200;
				ELSE
					fb_state_entry.i16_next_step := 210;
				END_IF
			END_IF
		END_IF

		IF fb_state_entry.X THEN
			gst_PersDaten.b_Zelle_nicht_in_Betrieb := FALSE;
		END_IF

(*=======================================================*)
	200:  (* Fahre Z-Achse bis auf 0-Koordinate des ISK - Y-Achse ist gekoppelt *)
		(* Einfahrhöhe der Y-Achse beachten! *)
		IF fb_state_entry.E THEN
			IF gst_datensatz.st_wkz.bFahreSofortAufUebergabePosition THEN
				fb_axis.lr_soll_geschwindigkeit := st_geschwindigkeiten.lr_auto_max;
			ELSE
				fb_axis.lr_soll_geschwindigkeit := gst_datensatz.st_wkz.r_auto_z;
			END_IF
			fb_axis.st_position.r_soll := gst_datensatz.st_isk.lr_pos_z_0 + gst_datensatz.st_wkz.lr_offset_z_pos_0 + gst_datensatz.st_wt.lr_offset_z_pos_0 + gst_datensatz.st_md.lr_offset_z_pos_0 + gst_datensatz.st_bestueckprogramm.lr_z[0];
			st_drive_cmd.enu_cmd := MOVE_ABSOLUTE;
			(*Rasterfolie kann gleich eingezogen werden. Zeitersparnis*)
			IF gst_datensatz.st_md.i16_typ_zelle = RASTERFOLIE THEN
				rasterfolieneinzug.st_ctrl.in.b_start := TRUE;
			END_IF
		END_IF

		(*-----------------------Weiterschaltbedingungen----------------------------*)
		(* Z-Achse losfahren und währenddessen beschreibt der Tagreader die Pille *)
		(*Rasterfolie kann gleich eingezogen werden. Zeitersparnis*)
		IF gst_datensatz.st_md.i16_typ_zelle = RASTERFOLIE THEN
			IF NOT rasterfolieneinzug.st_ctrl.out.b_fertig THEN
				rasterfolieneinzug.st_ctrl.in.b_start := FALSE;
				fb_state_entry.i16_next_step := 210;
			END_IF
		ELSE
			fb_state_entry.i16_next_step := 210;
		END_IF

(*=======================================================*)
	210:	(* WT als schlecht markieren *)
		IF fb_state_entry.E THEN
			ST_Markiere_WT_NIO();
		END_IF

		(*-----------------------Weiterschaltbedingungen----------------------------*)
		IF balluff_tag_reader.st_ctrl.out.b_fertig AND NOT fb_state_entry.E THEN
			(* Ok: Daten sind auf der Pille *)
			balluff_tag_reader.st_ctrl.in.b_start_schreiben := FALSE;
			IF gst_datensatz.st_md.b_tagreader_fahrend THEN
				(* Auf Z-Achse warten *)
				fb_state_entry.i16_next_step := 220;
			ELSE
				(* Daten geschrieben und erst jetzt die Z-Achse fahren *)
				fb_state_entry.i16_next_step := 230;
			END_IF
		END_IF

(*=======================================================*)
	220:	(* Warte noch auf die Z-Achse, bis sie im Ziel steht. *)

		(*-----------------------Weiterschaltbedingungen----------------------------*)
		IF st_drive_cmd.enu_cmd = NO_COMMAND THEN
			IF gst_datensatz.st_md.i16_typ_zelle = RASTERFOLIE THEN
				IF rasterfolieneinzug.st_ctrl.out.b_fertig THEN
					fb_state_entry.i16_next_step := 240;
				END_IF
			ELSE
				fb_state_entry.i16_next_step := 240;
			END_IF
		END_IF

(*=======================================================*)
	230:(* Fahre Z-Achse bis auf 0-Koordinate des ISK - Y-Achse ist gekoppelt *)
		(* Einfahrhöhe der Y-Achse beachten! *)
		IF fb_state_entry.E THEN
			(* Z-Achse verfahren*)
			IF gst_datensatz.st_wkz.bFahreSofortAufUebergabePosition THEN
				fb_axis.lr_soll_geschwindigkeit := st_geschwindigkeiten.lr_auto_max;
			ELSE
				fb_axis.lr_soll_geschwindigkeit := gst_datensatz.st_wkz.r_auto_z;
			END_IF
			fb_axis.st_position.r_soll := gst_datensatz.st_isk.lr_pos_z_0 + gst_datensatz.st_wkz.lr_offset_z_pos_0 + gst_datensatz.st_wt.lr_offset_z_pos_0 + gst_datensatz.st_md.lr_offset_z_pos_0 + gst_datensatz.st_bestueckprogramm.lr_z[0];
			st_drive_cmd.enu_cmd := MOVE_ABSOLUTE;
			(*Rasterfolie kann gleich eingezogen werden. Zeitersparnis*)
			IF gst_datensatz.st_md.i16_typ_zelle = RASTERFOLIE THEN
				rasterfolieneinzug.st_ctrl.in.b_start := TRUE;
			END_IF
		END_IF

		(*-----------------------Weiterschaltbedingungen----------------------------*)
		(* Z-Achse losfahren und währenddessen beschreibt der Tagreader die Pille *)
		(*Rasterfolie kann gleich eingezogen werden. Zeitersparnis*)
		IF gst_datensatz.st_md.i16_typ_zelle = RASTERFOLIE THEN
			IF NOT rasterfolieneinzug.st_ctrl.out.b_fertig THEN
				rasterfolieneinzug.st_ctrl.in.b_start := FALSE;
				fb_state_entry.i16_next_step := 235;
			END_IF
		ELSE
			fb_state_entry.i16_next_step := 235;
		END_IF

(*=======================================================*)
	235:	(* Warte noch auf die Z-Achse, bis sie im Ziel steht. *)

		(*-----------------------Weiterschaltbedingungen----------------------------*)
		IF st_drive_cmd.enu_cmd = NO_COMMAND THEN
			IF gst_datensatz.st_md.i16_typ_zelle = RASTERFOLIE THEN
				IF rasterfolieneinzug.st_ctrl.out.b_fertig THEN
					fb_state_entry.i16_next_step := 240;
				END_IF
			ELSE
				fb_state_entry.i16_next_step := 240;
			END_IF
		END_IF

(*=======================================================*)
	240:	(* Camout Y-Achse *)
		IF fb_state_entry.E THEN
			st_drive_cmd_y_achse.enu_cmd := CAM_OUT_SLAVE;
		END_IF

		(*-----------------------Weiterschaltbedingungen----------------------------*)
		IF st_drive_cmd_y_achse.enu_cmd = NO_COMMAND THEN
			fb_state_entry.i16_next_step := 250;
		END_IF

(*=======================================================*)
	250: (* Start Y-Achse positionieren auf  0-Koordinate  des ISK *)
		IF fb_state_entry.E THEN
			axis_y_achse.st_ctrl.in.b_start := TRUE;
		END_IF

		(*-----------------------Weiterschaltbedingungen----------------------------*)
		IF axis_y_achse.st_ctrl.out.b_fertig THEN	(* axis_y_achse.st_ctrl.out.b_busy  THEN *)
			fb_state_entry.i16_next_step := 255;
		END_IF

		IF fb_state_entry.X THEN
			axis_y_achse.st_ctrl.in.b_start := FALSE;
		END_IF

(*=======================================================*)
	255: (* Start Y-Achse positionieren auf  0-Koordinate  des ISK *)

		(*-----------------------Weiterschaltbedingungen----------------------------*)
		IF 	axis_y_achse.st_ctrl.out.b_fertig  THEN
			fb_state_entry.i16_next_step := 260;
		END_IF

(*=======================================================*)
	260:
		IF fb_state_entry.E THEN
			fb_Z_Achse_einfahren(b_start:= FALSE, t_zeit=> t_Z_Achse_einfahren);
			fb_Bestueckung(b_start:= TRUE, t_zeit=> );
		END_IF

		CASE gst_datensatz.st_md.i16_typ_zelle OF
			KEINE_ZELLE:
				;

			BESTUECKZELLE_1700:
				(* Führung wird an die Bestückachse abgegeben und die Z-Achse und Y-Achse wird ausschliesslich über Kurvenscheiben-Kopplung verfahren *)
				IF fb_state_entry.E THEN
					axis_virt_master.st_ctrl.in.b_start := TRUE;
				END_IF

				(*-----------------------Weiterschaltbedingungen----------------------------*)
				IF NOT axis_virt_master.st_ctrl.out.b_fertig THEN
					axis_virt_master.st_ctrl.in.b_start := FALSE;
					fb_state_entry.i16_next_step := 270;
				END_IF

			RASTERFOLIE:
				(* Starten der Rasterfolienmontagestation *)
				IF fb_state_entry.E THEN
					rasterfolienmontage.st_ctrl.in.b_start := TRUE;
				END_IF

				(*-----------------------Weiterschaltbedingungen----------------------------*)
				IF NOT rasterfolienmontage.st_ctrl.out.b_fertig THEN
					rasterfolienmontage.st_ctrl.in.b_start := FALSE;
					fb_state_entry.i16_next_step := 290;
				END_IF
		END_CASE

(*=======================================================*)
	270:	(* Bestückzelle 1700 *)

		(*-----------------------Weiterschaltbedingungen----------------------------*)
		IF axis_virt_master.st_ctrl.out.b_fertig THEN
			fb_state_entry.i16_next_step := 300;
		END_IF

		IF fb_state_entry.X THEN
			(* Stoppe Bestückzeit *)
			zeit_wt_bestuecken := TIME_TO_DWORD(fb_ton_taktzeitmessung_bestuecken.ET);
			fb_ton_taktzeitmessung_bestuecken.IN := FALSE;

			(* Starte WT Wechselzeit *)
			fb_ton_taktzeitmessung_wt_wechsel.IN := TRUE;
			fb_Bestueckung(b_start:= FALSE, t_zeit=>t_Bestueckung );
			fb_Z_Achse_ausfahren(b_start:= TRUE, t_zeit=> );
		END_IF

(*=======================================================*)
	290:	(* Rasterfolie *)

		(*-----------------------Weiterschaltbedingungen----------------------------*)
		IF 	rasterfolienmontage.st_ctrl.out.b_fertig THEN
			fb_state_entry.i16_next_step := 294;
		END_IF

		IF fb_state_entry.X THEN
			(* Stoppe Bestückzeit *)
			zeit_wt_bestuecken := TIME_TO_DWORD(fb_ton_taktzeitmessung_bestuecken.ET);
			fb_ton_taktzeitmessung_bestuecken.IN := FALSE;
			(* Starte WT Wechselzeit *)
			fb_ton_taktzeitmessung_wt_wechsel.IN := TRUE;
			fb_Bestueckung(b_start:= FALSE, t_zeit=>t_Bestueckung );
			fb_Z_Achse_ausfahren(b_start:= TRUE, t_zeit=> );
		END_IF

(*=======================================================*)
	294:(* Fahre Z-Achse auf  Rasterfolienprüfposition *)
		IF fb_state_entry.E THEN


			(* Z-Achse verfahren*)
			fb_axis.lr_soll_geschwindigkeit := gst_datensatz.st_wkz.r_auto_z;
			fb_axis.st_position.r_soll := 	gst_datensatz.st_isk.lr_pos_z_0 + gst_datensatz.st_wkz.lr_offset_z_pos_0 + gst_datensatz.st_wt.lr_offset_z_pos_0 + gst_datensatz.st_md.lr_offset_z_pos_0 + gst_datensatz.st_bestueckprogramm.lr_z[i32_anzahl_rasterfolie] +	(*Bestückposition*)
										gst_datensatz.st_wkz.st_rasterfolie.lr_pruefpos_rafo;	(*Abstand zwischen Bestückposition und Prüfposition*)
			st_drive_cmd.enu_cmd := MOVE_ABSOLUTE;
		END_IF

		(*-----------------------Weiterschaltbedingungen----------------------------*)
		IF 	st_drive_cmd.enu_cmd = NO_COMMAND AND
			ST_Rasterfolienmontage.arr_rafo_schieberegister[i32_anzahl_rasterfolie] THEN (*Folie vorhanden*)
			fb_state_entry.i16_next_step := 296;
		END_IF

(*=======================================================*)
	296:	(* Anzahl der Rasterfolien prüfen*)

		IF 	fb_state_entry.E THEN
			i32_anzahl_rasterfolie:=i32_anzahl_rasterfolie+1;
		END_IF

		(*-----------------------Weiterschaltbedingungen----------------------------*)
		IF 	i32_anzahl_rasterfolie = gst_datensatz.st_bestueckprogramm.i32_anzahl THEN
			fb_state_entry.i16_next_step := 300;	 (*Ende*)
		ELSE
			fb_state_entry.i16_next_step := 297;	 (*zur nächsten Folie*)
		END_IF

(*=======================================================*)
	297:(* Fahre Z-Achse auf nächste Rasterfolienposition *)
		IF 	fb_state_entry.E THEN
			(* Z-Achse verfahren*)
			fb_axis.lr_soll_geschwindigkeit := gst_datensatz.st_wkz.r_auto_z;
			fb_axis.st_position.r_soll := gst_datensatz.st_isk.lr_pos_z_0 + gst_datensatz.st_wkz.lr_offset_z_pos_0 + gst_datensatz.st_wt.lr_offset_z_pos_0 + gst_datensatz.st_md.lr_offset_z_pos_0 + gst_datensatz.st_bestueckprogramm.lr_z[i32_anzahl_rasterfolie];
			st_drive_cmd.enu_cmd := MOVE_ABSOLUTE;
		END_IF

		(*-----------------------Weiterschaltbedingungen----------------------------*)
		IF st_drive_cmd.enu_cmd = NO_COMMAND THEN
			fb_state_entry.i16_next_step := 298;
		END_IF

(*=======================================================*)
	298:(* Fahre Z-Achse auf nächste Rasterfolienposition *)
		IF 	fb_state_entry.E THEN
			(*Rasterfolie kann gleich eingezogen werden. Zeitersparnis*)
			rasterfolieneinzug.st_ctrl.in.b_start := TRUE;
		END_IF

		(*-----------------------Weiterschaltbedingungen----------------------------*)
		(* Z-Achse losfahren und währenddessen beschreibt der Tagreader die Pille *)
		(*Rasterfolie kann gleich eingezogen werden. Zeitersparnis*)
		IF NOT rasterfolieneinzug.st_ctrl.out.b_fertig THEN
			rasterfolieneinzug.st_ctrl.in.b_start := FALSE;
			fb_state_entry.i16_next_step := 299;
		END_IF

(*=======================================================*)
	299:	(* Neue Folie eingezogen. *)

		(*-----------------------Weiterschaltbedingungen----------------------------*)
		IF rasterfolieneinzug.st_ctrl.out.b_fertig THEN
			fb_state_entry.i16_next_step := 240;	(*zurück zum nächsten Folien setzen*)
		END_IF

(*=======================================================*)
	300: (* Auslesen der Y-Position an der aktuellen Z-Position in der Kurvenscheibe *)
		IF 	fb_state_entry.E THEN
			fb_axis_y_achse.r_master_position := z_achse.NcToPlc.ActPos;
			st_drive_cmd_y_achse.enu_cmd := READ_SLAVE_DYNAMICS;
		END_IF

		(*-----------------------Weiterschaltbedingungen----------------------------*)
		IF 	st_drive_cmd_y_achse.enu_cmd = NO_COMMAND THEN
			fb_state_entry.i16_next_step := 310;
		END_IF

(*=======================================================*)
	310: (* Start Y-Achse positionieren zurück auf die Kurvenbahn *)
		IF 	fb_state_entry.E THEN
			lr_slave_position := fb_axis_y_achse.mc_read_camtable_slave_dynamics.SlavePosition;
			axis_y_achse.st_ctrl.in.b_start_2 := TRUE;
		END_IF

		(*-----------------------Weiterschaltbedingungen----------------------------*)
		IF axis_y_achse.st_ctrl.out.b_fertig_2 AND NOT fb_state_entry.E THEN
			axis_y_achse.st_ctrl.in.b_start_2 := FALSE;
			fb_state_entry.i16_next_step := 315;
		END_IF

(*=======================================================*)
	315: (* Abfrage, ob sofort auf Übergabeposition gefahren werden soll *)

		(*-----------------------Weiterschaltbedingungen----------------------------*)
		IF gst_datensatz.st_wkz.bFahreSofortAufUebergabePosition THEN
			fb_state_entry.i16_next_step := 330;
		ELSE
			fb_state_entry.i16_next_step := 320;
		END_IF

(*=======================================================*)
	320:	(* Fahre Z-Achse bis auf Anfang der Kurvenbahn *)
		IF fb_state_entry.E THEN
			fb_axis.lr_soll_geschwindigkeit := st_geschwindigkeiten.lr_auto_max;
			IF gst_datensatz.st_wkz.b_variable_einfahrposition THEN
				fb_axis.st_position.r_soll := gst_datensatz.st_wkz.st_yz_tisch.r_wkz_einfahrpos_z;
			ELSE
				fb_axis.st_position.r_soll := ST_MotionFunctionPoints.YZTischMasterPos2;
			END_IF
			st_drive_cmd.enu_cmd := MOVE_ABSOLUTE;
		END_IF

		(*-----------------------Weiterschaltbedingungen----------------------------*)
		IF st_drive_cmd.enu_cmd = NO_COMMAND THEN
			fb_state_entry.i16_next_step := 330;
		END_IF

(*=======================================================*)
	330:	(* Camin Y-Achse *)
		IF fb_state_entry.E THEN
			fb_axis_y_achse.st_camscaling_data.SlaveScaling := 1;
			st_drive_cmd_y_achse.enu_cmd := CAM_IN_SLAVE;
		END_IF

		(*-----------------------Weiterschaltbedingungen----------------------------*)
		IF st_drive_cmd_y_achse.enu_cmd = NO_COMMAND THEN
			fb_state_entry.i16_next_step := 340;
		END_IF

(*=======================================================*)
	340:	(* Fahre Z-Achse mit gekoppelter Y-Achse bis auf Übergabeposition *)
		IF fb_state_entry.E THEN
			IF gst_datensatz.st_wkz.bFahreSofortAufUebergabePosition THEN
				fb_axis.lr_soll_geschwindigkeit := st_geschwindigkeiten.lr_auto_max;
			ELSE
				fb_axis.lr_soll_geschwindigkeit := gst_datensatz.st_wkz.r_auto_z;
			END_IF
			fb_axis.st_position.r_soll := gst_datensatz.st_md.st_md_z_achse.lr_wt_uebergabepos;
			st_drive_cmd.enu_cmd := MOVE_ABSOLUTE;
		END_IF

		(*Nach einem Bandwechsel soll nach X-Teilen gestoppt werden.*)
		IF gst_datensatz.st_wkz.i16_anzahl_Teile_autostop_bandwechsel > 0 THEN
			IF gi16_anzahl_Teile_autostop_bandwechsel = gst_datensatz.st_wkz.i16_anzahl_Teile_autostop_bandwechsel THEN
				Teile_nach_Bandwechsel := TRUE;
				gb_nach_bawe_einzelfertigung := TRUE;
			END_IF
		END_IF

